LIN {X 0,Y 523.484,Z 545.078,A -85,B 0,C 180,E1 -4763.834,E2 -4763.834} C_VEL
LIN {X 0,Y 523.383,Z 549.826,A -85,B 0,C 180,E1 -4764.992,E2 -4764.992} C_VEL
LIN {X 0,Y 523.443,Z 553.457,A -85,B 0,C 180,E1 -4766.15,E2 -4766.15} C_VEL
LIN {X 0,Y 523.367,Z 555.329,A -85,B 0,C 180,E1 -4766.921,E2 -4766.921} C_VEL
LIN {X 0,Y 523.334,Z 556.731,A -85,B 0,C 180,E1 -4767.691,E2 -4767.691} C_VEL
LIN {X 0,Y 523.25,Z 558.341,A -85,B 0,C 180,E1 -4769.23,E2 -4769.23} C_VEL
LIN {X 0,Y 523.25,Z 558.562,A -85,B 0,C 180,E1 -4770,E2 -4770} C_VEL
LIN {X 0,Y 523.274,Z 557.74,A -85,B 0,C 180,E1 -4771.539,E2 -4771.539} C_VEL
LIN {X 0,Y 523.334,Z 556.745,A -85,B 0,C 180,E1 -4772.308,E2 -4772.308} C_VEL
LIN {X 0,Y 523.367,Z 555.347,A -85,B 0,C 180,E1 -4773.079,E2 -4773.079} C_VEL
LIN {X 0,Y 523.424,Z 552.405,A -85,B 0,C 180,E1 -4774.235,E2 -4774.235} C_VEL
LIN {X 0,Y 523.461,Z 548.419,A -85,B 0,C 180,E1 -4775.392,E2 -4775.392} C_VEL
LIN {X 0,Y 523.514,Z 543.187,A -85,B 0,C 180,E1 -4776.572,E2 -4776.572} C_VEL
LIN {X 0,Y 523.638,Z 536.823,A -85,B 0,C 180,E1 -4777.713,E2 -4777.713} C_VEL
LIN {X 0,Y 523.814,Z 528.761,A -85,B 0,C 180,E1 -4778.875,E2 -4778.875} C_VEL
LIN {X 0,Y 524.041,Z 520.543,A -85,B 0,C 180,E1 -4779.845,E2 -4779.845} C_VEL
LIN {X 0,Y 524.298,Z 510.517,A -85,B 0,C 180,E1 -4780.816,E2 -4780.816} C_VEL
LIN {X 0,Y 524.6,Z 499.164,A -85,B 0,C 180,E1 -4781.691,E2 -4781.691} C_VEL
LIN {X 0,Y 524.837,Z 488.067,A -85,B 0,C 180,E1 -4782.371,E2 -4782.371} C_VEL
LIN {X 0,Y 525.075,Z 475.733,A -85,B 0,C 180,E1 -4782.955,E2 -4782.955} C_VEL
LIN {X 0,Y 525.31,Z 462.663,A -85,B 0,C 180,E1 -4783.392,E2 -4783.392} C_VEL
LIN {X 0,Y 525.513,Z 450.182,A -85,B 0,C 180,E1 -4783.658,E2 -4783.658} C_VEL
LIN {X 0,Y 525.797,Z 355.668,A -85,B 0,C 180,E1 -4784.969,E2 -4784.969} C_VEL
LIN {X 0,Y 524.316,Z 345.731,A -85,B 0,C 180,E1 -4785.168,E2 -4785.168} C_VEL
LIN {X 0,Y 524.755,Z 323.816,A -85,B 0,C 180,E1 -4788.526,E2 -4788.526} C_VEL
LIN {X 0,Y 525.188,Z 305.323,A -85,B 0,C 180,E1 -4791.386,E2 -4791.386} C_VEL
LIN {X 0,Y 525.479,Z 293.613,A -85,B 0,C 180,E1 -4793.237,E2 -4793.237} C_VEL
LIN {X 0,Y 523.982,Z 285.216,A -85,B 0,C 180,E1 -4794.674,E2 -4794.674} C_VEL
LIN {X 0,Y 523.978,Z 285.218,A -85,B 0,C 180,E1 -4797.718,E2 -4797.718} C_VEL
LIN {X 0,Y 523.943,Z 285.215,A -85,B 0,C 180,E1 -4800.854,E2 -4800.854} C_VEL
LIN {X 0,Y 523.957,Z 285.216,A -85,B 0,C 180,E1 -4803.734,E2 -4803.734} C_VEL
LIN {X 0,Y 523.901,Z 285.227,A -85,B 0,C 180,E1 -4806.401,E2 -4806.401} C_VEL
LIN {X 0,Y 523.917,Z 285.218,A -85,B 0,C 180,E1 -4809.084,E2 -4809.084} C_VEL
LIN {X 0,Y 523.952,Z 285.218,A -85,B 0,C 180,E1 -4812.118,E2 -4812.118} C_VEL
LIN {X 0,Y 523.952,Z 285.213,A -85,B 0,C 180,E1 -4815.308,E2 -4815.308} C_VEL
LIN {X 0,Y 523.958,Z 285.221,A -85,B 0,C 180,E1 -4818.688,E2 -4818.688} C_VEL
LIN {X 0,Y 523.915,Z 285.218,A -85,B 0,C 180,E1 -4821.898,E2 -4821.898} C_VEL
LIN {X 0,Y 523.93,Z 285.224,A -85,B 0,C 180,E1 -4824.909,E2 -4824.909} C_VEL
LIN {X 0,Y 523.938,Z 285.215,A -85,B 0,C 180,E1 -4827.678,E2 -4827.678} C_VEL
LIN {X 0,Y 523.949,Z 285.219,A -85,B 0,C 180,E1 -4830.676,E2 -4830.676} C_VEL
LIN {X 0,Y 523.969,Z 285.212,A -85,B 0,C 180,E1 -4833.728,E2 -4833.728} C_VEL
LIN {X 0,Y 523.931,Z 285.216,A -85,B 0,C 180,E1 -4836.271,E2 -4836.271} C_VEL
LIN {X 0,Y 523.94,Z 285.219,A -85,B 0,C 180,E1 -4838.766,E2 -4838.766} C_VEL
LIN {X 0,Y 523.946,Z 285.224,A -85,B 0,C 180,E1 -4841.221,E2 -4841.221} C_VEL
LIN {X 0,Y 523.931,Z 285.22,A -85,B 0,C 180,E1 -4843.639,E2 -4843.639} C_VEL
LIN {X 0,Y 523.939,Z 285.216,A -85,B 0,C 180,E1 -4846.028,E2 -4846.028} C_VEL
LIN {X 0,Y 524.006,Z 285.206,A -85,B 0,C 180,E1 -4848.394,E2 -4848.394} C_VEL
LIN {X 0,Y 523.999,Z 285.217,A -85,B 0,C 180,E1 -4851.516,E2 -4851.516} C_VEL
LIN {X 0,Y 524.077,Z 285.198,A -85,B 0,C 180,E1 -4854.614,E2 -4854.614} C_VEL
LIN {X 0,Y 524.103,Z 285.204,A -85,B 0,C 180,E1 -4857.695,E2 -4857.695} C_VEL
LIN {X 0,Y 524.116,Z 285.193,A -85,B 0,C 180,E1 -4860.769,E2 -4860.769} C_VEL
LIN {X 0,Y 524.067,Z 285.2,A -85,B 0,C 180,E1 -4863.075,E2 -4863.075} C_VEL
LIN {X 0,Y 524.023,Z 285.21,A -85,B 0,C 180,E1 -4866.16,E2 -4866.16} C_VEL
LIN {X 0,Y 523.998,Z 285.21,A -85,B 0,C 180,E1 -4868.484,E2 -4868.484} C_VEL
LIN {X 0,Y 523.997,Z 285.213,A -85,B 0,C 180,E1 -4871.74,E2 -4871.74} C_VEL
LIN {X 0,Y 523.986,Z 285.209,A -85,B 0,C 180,E1 -4875.052,E2 -4875.052} C_VEL
LIN {X 0,Y 523.942,Z 285.22,A -85,B 0,C 180,E1 -4877.97,E2 -4877.97} C_VEL
LIN {X 0,Y 523.967,Z 285.219,A -85,B 0,C 180,E1 -4880.411,E2 -4880.411} C_VEL
LIN {X 0,Y 523.905,Z 285.221,A -85,B 0,C 180,E1 -4882.894,E2 -4882.894} C_VEL
LIN {X 0,Y 523.925,Z 285.216,A -85,B 0,C 180,E1 -4885.42,E2 -4885.42} C_VEL
LIN {X 0,Y 523.913,Z 285.221,A -85,B 0,C 180,E1 -4888.003,E2 -4888.003} C_VEL
LIN {X 0,Y 523.94,Z 285.22,A -85,B 0,C 180,E1 -4890.855,E2 -4890.855} C_VEL
LIN {X 0,Y 523.955,Z 285.213,A -85,B 0,C 180,E1 -4893.735,E2 -4893.735} C_VEL
LIN {X 0,Y 523.9,Z 285.225,A -85,B 0,C 180,E1 -4896.402,E2 -4896.402} C_VEL
LIN {X 0,Y 523.91,Z 285.223,A -85,B 0,C 180,E1 -4899.086,E2 -4899.086} C_VEL
LIN {X 0,Y 523.935,Z 285.216,A -85,B 0,C 180,E1 -4902.121,E2 -4902.121} C_VEL
LIN {X 0,Y 523.938,Z 285.219,A -85,B 0,C 180,E1 -4905.311,E2 -4905.311} C_VEL
LIN {X 0,Y 523.894,Z 285.227,A -85,B 0,C 180,E1 -4906.894,E2 -4906.894} C_VEL
LIN {X 0,Y 523.214,Z 285.308,A -85,B 0,C 180,E1 -4907.535,E2 -4907.535} C_VEL
LIN {X 0,Y 520.363,Z 285.663,A -85,B 0,C 180,E1 -4908.577,E2 -4908.577} C_VEL
LIN {X 0,Y 517.964,Z 285.963,A -85,B 0,C 180,E1 -4909.416,E2 -4909.416} C_VEL
LIN {X 0,Y 516.939,Z 286.087,A -85,B 0,C 180,E1 -4910.063,E2 -4910.063} C_VEL
LIN {X 0,Y 516.857,Z 286.097,A -85,B 0,C 180,E1 -4910.283,E2 -4910.283} C_VEL
LIN {X 0,Y 516.874,Z 286.104,A -85,B 0,C 180,E1 -4913.255,E2 -4913.255} C_VEL
LIN {X 0,Y 516.884,Z 286.094,A -85,B 0,C 180,E1 -4916.12,E2 -4916.12} C_VEL
LIN {X 0,Y 516.88,Z 286.098,A -85,B 0,C 180,E1 -4918.939,E2 -4918.939} C_VEL
LIN {X 0,Y 516.849,Z 286.105,A -85,B 0,C 180,E1 -4921.581,E2 -4921.581} C_VEL
LIN {X 0,Y 516.86,Z 286.097,A -85,B 0,C 180,E1 -4924.208,E2 -4924.208} C_VEL
LIN {X 0,Y 516.859,Z 286.097,A -85,B 0,C 180,E1 -4926.777,E2 -4926.777} C_VEL
LIN {X 0,Y 516.933,Z 286.096,A -85,B 0,C 180,E1 -4929.735,E2 -4929.735} C_VEL
LIN {X 0,Y 516.887,Z 286.093,A -85,B 0,C 180,E1 -4932.595,E2 -4932.595} C_VEL
LIN {X 0,Y 516.946,Z 286.087,A -85,B 0,C 180,E1 -4935.031,E2 -4935.031} C_VEL
LIN {X 0,Y 516.93,Z 286.092,A -85,B 0,C 180,E1 -4938.233,E2 -4938.233} C_VEL
LIN {X 0,Y 516.923,Z 286.091,A -85,B 0,C 180,E1 -4941.399,E2 -4941.399} C_VEL
LIN {X 0,Y 516.983,Z 286.084,A -85,B 0,C 180,E1 -4944.54,E2 -4944.54} C_VEL
LIN {X 0,Y 517.071,Z 286.073,A -85,B 0,C 180,E1 -4947.664,E2 -4947.664} C_VEL
LIN {X 0,Y 517.068,Z 286.078,A -85,B 0,C 180,E1 -4950,E2 -4950} C_VEL
LIN {X 0,Y 517.069,Z 286.079,A -85,B 0,C 180,E1 -4952.337,E2 -4952.337} C_VEL
LIN {X 0,Y 516.972,Z 286.091,A -85,B 0,C 180,E1 -4956.244,E2 -4956.244} C_VEL
LIN {X 0,Y 516.902,Z 286.091,A -85,B 0,C 180,E1 -4959.391,E2 -4959.391} C_VEL
LIN {X 0,Y 516.882,Z 286.103,A -85,B 0,C 180,E1 -4962.566,E2 -4962.566} C_VEL
LIN {X 0,Y 516.837,Z 286.1,A -85,B 0,C 180,E1 -4965.781,E2 -4965.781} C_VEL
LIN {X 0,Y 516.874,Z 286.098,A -85,B 0,C 180,E1 -4968.224,E2 -4968.224} C_VEL
LIN {X 0,Y 516.882,Z 286.103,A -85,B 0,C 180,E1 -4970.703,E2 -4970.703} C_VEL
LIN {X 0,Y 516.848,Z 286.104,A -85,B 0,C 180,E1 -4973.225,E2 -4973.225} C_VEL
LIN {X 0,Y 516.856,Z 286.102,A -85,B 0,C 180,E1 -4976.175,E2 -4976.175} C_VEL
LIN {X 0,Y 516.912,Z 286.308,A -85,B 0,C 180,E1 -4977.15,E2 -4977.15} C_VEL
LIN {X 0,Y 517.552,Z 290.673,A -85,B 0,C 180,E1 -4978.035,E2 -4978.035} C_VEL
LIN {X 0,Y 517.288,Z 305.162,A -85,B 0,C 180,E1 -4980.856,E2 -4980.856} C_VEL
LIN {X 0,Y 517.209,Z 309.487,A -85,B 0,C 180,E1 -4981.687,E2 -4981.687} C_VEL
LIN {X 0,Y 519.12,Z 321.055,A -85,B 0,C 180,E1 -4981.925,E2 -4981.925} C_VEL
LIN {X 0,Y 518.626,Z 416.658,A -85,B 0,C 180,E1 -4983.288,E2 -4983.288} C_VEL
LIN {X 0,Y 518.388,Z 430.021,A -85,B 0,C 180,E1 -4983.641,E2 -4983.641} C_VEL
LIN {X 0,Y 518.174,Z 441.438,A -85,B 0,C 180,E1 -4984.086,E2 -4984.086} C_VEL
LIN {X 0,Y 517.884,Z 452.681,A -85,B 0,C 180,E1 -4984.668,E2 -4984.668} C_VEL
LIN {X 0,Y 517.613,Z 463.334,A -85,B 0,C 180,E1 -4985.369,E2 -4985.369} C_VEL
LIN {X 0,Y 517.364,Z 473.747,A -85,B 0,C 180,E1 -4986.222,E2 -4986.222} C_VEL
LIN {X 0,Y 517.004,Z 484.69,A -85,B 0,C 180,E1 -4987.346,E2 -4987.346} C_VEL
LIN {X 0,Y 516.8,Z 492.236,A -85,B 0,C 180,E1 -4988.305,E2 -4988.305} C_VEL
LIN {X 0,Y 516.619,Z 499.468,A -85,B 0,C 180,E1 -4989.426,E2 -4989.426} C_VEL
LIN {X 0,Y 516.474,Z 504.474,A -85,B 0,C 180,E1 -4990.356,E2 -4990.356} C_VEL
LIN {X 0,Y 516.39,Z 509.598,A -85,B 0,C 180,E1 -4991.535,E2 -4991.535} C_VEL
LIN {X 0,Y 516.329,Z 513.522,A -85,B 0,C 180,E1 -4992.69,E2 -4992.69} C_VEL
LIN {X 0,Y 516.259,Z 516.694,A -85,B 0,C 180,E1 -4993.97,E2 -4993.97} C_VEL
LIN {X 0,Y 516.213,Z 518.527,A -85,B 0,C 180,E1 -4995.069,E2 -4995.069} C_VEL
LIN {X 0,Y 516.184,Z 519.573,A -85,B 0,C 180,E1 -4996.188,E2 -4996.188} C_VEL
LIN {X 0,Y 516.178,Z 519.794,A -85,B 0,C 180,E1 -4997.327,E2 -4997.327} C_VEL
LIN {X 0,Y 516.197,Z 519.147,A -85,B 0,C 180,E1 -4998.489,E2 -4998.489} C_VEL
LIN {X 0,Y 516.196,Z 517.568,A -85,B 0,C 180,E1 -4999.68,E2 -4999.68} C_VEL
LIN {X 0,Y 516.287,Z 514.031,A -85,B 0,C 180,E1 -5001.231,E2 -5001.231} C_VEL
LIN {X 0,Y 516.386,Z 510.828,A -85,B 0,C 180,E1 -5002.233,E2 -5002.233} C_VEL
LIN {X 0,Y 516.471,Z 506.049,A -85,B 0,C 180,E1 -5003.404,E2 -5003.404} C_VEL
LIN {X 0,Y 516.586,Z 500.555,A -85,B 0,C 180,E1 -5004.483,E2 -5004.483} C_VEL
LIN {X 0,Y 516.783,Z 493.342,A -85,B 0,C 180,E1 -5005.634,E2 -5005.634} C_VEL
LIN {X 0,Y 517.017,Z 485.983,A -85,B 0,C 180,E1 -5006.596,E2 -5006.596} C_VEL
LIN {X 0,Y 517.277,Z 476.668,A -85,B 0,C 180,E1 -5007.603,E2 -5007.603} C_VEL
LIN {X 0,Y 517.538,Z 465.559,A -85,B 0,C 180,E1 -5008.562,E2 -5008.562} C_VEL
LIN {X 0,Y 517.86,Z 454.909,A -85,B 0,C 180,E1 -5009.295,E2 -5009.295} C_VEL
LIN {X 0,Y 518.163,Z 442.997,A -85,B 0,C 180,E1 -5009.935,E2 -5009.935} C_VEL
LIN {X 0,Y 518.359,Z 430.294,A -85,B 0,C 180,E1 -5010.442,E2 -5010.442} C_VEL
LIN {X 0,Y 518.56,Z 416.327,A -85,B 0,C 180,E1 -5010.811,E2 -5010.811} C_VEL
LIN {X 0,Y 518.973,Z 319.058,A -85,B 0,C 180,E1 -5012.201,E2 -5012.201} C_VEL
LIN {X 0,Y 517.197,Z 309.037,A -85,B 0,C 180,E1 -5012.401,E2 -5012.401} C_VEL
LIN {X 0,Y 517.21,Z 289.506,A -85,B 0,C 180,E1 -5015.666,E2 -5015.666} C_VEL
LIN {X 0,Y 516.991,Z 286.087,A -85,B 0,C 180,E1 -5016.251,E2 -5016.251} C_VEL
LIN {X 0,Y 516.942,Z 286.092,A -85,B 0,C 180,E1 -5019.731,E2 -5019.731} C_VEL
LIN {X 0,Y 516.909,Z 286.095,A -85,B 0,C 180,E1 -5022.595,E2 -5022.595} C_VEL
LIN {X 0,Y 516.954,Z 286.092,A -85,B 0,C 180,E1 -5025.03,E2 -5025.03} C_VEL
LIN {X 0,Y 516.968,Z 286.085,A -85,B 0,C 180,E1 -5028.233,E2 -5028.233} C_VEL
LIN {X 0,Y 516.964,Z 286.091,A -85,B 0,C 180,E1 -5031.399,E2 -5031.399} C_VEL
LIN {X 0,Y 517.003,Z 286.088,A -85,B 0,C 180,E1 -5033.757,E2 -5033.757} C_VEL
LIN {X 0,Y 517.013,Z 286.079,A -85,B 0,C 180,E1 -5036.883,E2 -5036.883} C_VEL
LIN {X 0,Y 517.087,Z 286.077,A -85,B 0,C 180,E1 -5040,E2 -5040} C_VEL
LIN {X 0,Y 517.013,Z 286.078,A -85,B 0,C 180,E1 -5043.117,E2 -5043.117} C_VEL
LIN {X 0,Y 516.989,Z 286.087,A -85,B 0,C 180,E1 -5046.243,E2 -5046.243} C_VEL
LIN {X 0,Y 516.967,Z 286.087,A -85,B 0,C 180,E1 -5048.6,E2 -5048.6} C_VEL
LIN {X 0,Y 516.953,Z 286.088,A -85,B 0,C 180,E1 -5051.807,E2 -5051.807} C_VEL
LIN {X 0,Y 516.949,Z 286.087,A -85,B 0,C 180,E1 -5055.147,E2 -5055.147} C_VEL
LIN {X 0,Y 516.917,Z 286.093,A -85,B 0,C 180,E1 -5058.222,E2 -5058.222} C_VEL
LIN {X 0,Y 516.914,Z 286.096,A -85,B 0,C 180,E1 -5060.701,E2 -5060.701} C_VEL
LIN {X 0,Y 516.904,Z 286.092,A -85,B 0,C 180,E1 -5064.072,E2 -5064.072} C_VEL
LIN {X 0,Y 516.925,Z 286.096,A -85,B 0,C 180,E1 -5066.658,E2 -5066.658} C_VEL
LIN {X 0,Y 516.912,Z 286.092,A -85,B 0,C 180,E1 -5069.524,E2 -5069.524} C_VEL
LIN {X 0,Y 516.895,Z 286.095,A -85,B 0,C 180,E1 -5072.543,E2 -5072.543} C_VEL
LIN {X 0,Y 516.867,Z 286.103,A -85,B 0,C 180,E1 -5075.329,E2 -5075.329} C_VEL
LIN {X 0,Y 516.882,Z 286.094,A -85,B 0,C 180,E1 -5077.943,E2 -5077.943} C_VEL
LIN {X 0,Y 516.885,Z 286.096,A -85,B 0,C 180,E1 -5080.742,E2 -5080.742} C_VEL
LIN {X 0,Y 516.884,Z 286.098,A -85,B 0,C 180,E1 -5082.831,E2 -5082.831} C_VEL
LIN {X 0,Y 516.897,Z 286.097,A -85,B 0,C 180,E1 -5085.007,E2 -5085.007} C_VEL
LIN {X 0,Y 516.915,Z 286.091,A -85,B 0,C 180,E1 -5088.399,E2 -5088.399} C_VEL
LIN {X 0,Y 516.882,Z 286.1,A -85,B 0,C 180,E1 -5091.284,E2 -5091.284} C_VEL
LIN {X 0,Y 516.873,Z 286.101,A -85,B 0,C 180,E1 -5094.22,E2 -5094.22} C_VEL
LIN {X 0,Y 516.897,Z 286.097,A -85,B 0,C 180,E1 -5097.053,E2 -5097.053} C_VEL
LIN {X 0,Y 516.895,Z 286.102,A -85,B 0,C 180,E1 -5099.796,E2 -5099.796} C_VEL
LIN {X 0,Y 516.927,Z 286.095,A -85,B 0,C 180,E1 -5102.467,E2 -5102.467} C_VEL
LIN {X 0,Y 516.908,Z 286.098,A -85,B 0,C 180,E1 -5105.396,E2 -5105.396} C_VEL
LIN {X 0,Y 516.921,Z 286.184,A -85,B 0,C 180,E1 -5105.518,E2 -5105.518} C_VEL
LIN {X 0,Y 518.271,Z 294.325,A -85,B 0,C 180,E1 -5106.843,E2 -5106.843} C_VEL
LIN {X 0,Y 517.895,Z 313.462,A -85,B 0,C 180,E1 -5109.794,E2 -5109.794} C_VEL
LIN {X 0,Y 517.504,Z 331.908,A -85,B 0,C 180,E1 -5112.616,E2 -5112.616} C_VEL
LIN {X 0,Y 517.251,Z 345.235,A -85,B 0,C 180,E1 -5114.634,E2 -5114.634} C_VEL
LIN {X 0,Y 519.038,Z 358.299,A -85,B 0,C 180,E1 -5114.876,E2 -5114.876} C_VEL
LIN {X 0,Y 518.533,Z 453.585,A -85,B 0,C 180,E1 -5116.229,E2 -5116.229} C_VEL
LIN {X 0,Y 518.3,Z 466.903,A -85,B 0,C 180,E1 -5116.572,E2 -5116.572} C_VEL
LIN {X 0,Y 518.025,Z 479.679,A -85,B 0,C 180,E1 -5117.064,E2 -5117.064} C_VEL
LIN {X 0,Y 517.775,Z 491.966,A -85,B 0,C 180,E1 -5117.713,E2 -5117.713} C_VEL
LIN {X 0,Y 517.486,Z 504.066,A -85,B 0,C 180,E1 -5118.543,E2 -5118.543} C_VEL
LIN {X 0,Y 517.159,Z 514.372,A -85,B 0,C 180,E1 -5119.428,E2 -5119.428} C_VEL
LIN {X 0,Y 516.89,Z 523.628,A -85,B 0,C 180,E1 -5120.412,E2 -5120.412} C_VEL
LIN {X 0,Y 516.656,Z 532.638,A -85,B 0,C 180,E1 -5121.591,E2 -5121.591} C_VEL
LIN {X 0,Y 516.505,Z 539.895,A -85,B 0,C 180,E1 -5122.769,E2 -5122.769} C_VEL
LIN {X 0,Y 516.397,Z 544.787,A -85,B 0,C 180,E1 -5123.749,E2 -5123.749} C_VEL
LIN {X 0,Y 516.313,Z 549.544,A -85,B 0,C 180,E1 -5124.924,E2 -5124.924} C_VEL
LIN {X 0,Y 516.352,Z 553.181,A -85,B 0,C 180,E1 -5126.097,E2 -5126.097} C_VEL
LIN {X 0,Y 516.282,Z 555.056,A -85,B 0,C 180,E1 -5126.878,E2 -5126.878} C_VEL
LIN {X 0,Y 516.26,Z 556.462,A -85,B 0,C 180,E1 -5127.659,E2 -5127.659} C_VEL
LIN {X 0,Y 516.16,Z 558.076,A -85,B 0,C 180,E1 -5129.219,E2 -5129.219} C_VEL
LIN {X 0,Y 516.158,Z 558.298,A -85,B 0,C 180,E1 -5130,E2 -5130} C_VEL
LIN {X 0,Y 516.191,Z 557.476,A -85,B 0,C 180,E1 -5131.56,E2 -5131.56} C_VEL
LIN {X 0,Y 516.26,Z 556.482,A -85,B 0,C 180,E1 -5132.34,E2 -5132.34} C_VEL
LIN {X 0,Y 516.282,Z 555.082,A -85,B 0,C 180,E1 -5133.121,E2 -5133.121} C_VEL
LIN {X 0,Y 516.311,Z 552.137,A -85,B 0,C 180,E1 -5134.293,E2 -5134.293} C_VEL
LIN {X 0,Y 516.375,Z 548.148,A -85,B 0,C 180,E1 -5135.466,E2 -5135.466} C_VEL
LIN {X 0,Y 516.45,Z 542.212,A -85,B 0,C 180,E1 -5136.798,E2 -5136.798} C_VEL
LIN {X 0,Y 516.594,Z 535.298,A -85,B 0,C 180,E1 -5138.015,E2 -5138.015} C_VEL
LIN {X 0,Y 516.791,Z 526.97,A -85,B 0,C 180,E1 -5139.194,E2 -5139.194} C_VEL
LIN {X 0,Y 517.024,Z 518.423,A -85,B 0,C 180,E1 -5140.178,E2 -5140.178} C_VEL
LIN {X 0,Y 517.365,Z 507.866,A -85,B 0,C 180,E1 -5141.161,E2 -5141.161} C_VEL
LIN {X 0,Y 517.668,Z 496.325,A -85,B 0,C 180,E1 -5142.024,E2 -5142.024} C_VEL
LIN {X 0,Y 517.915,Z 485.935,A -85,B 0,C 180,E1 -5142.639,E2 -5142.639} C_VEL
LIN {X 0,Y 518.169,Z 474.071,A -85,B 0,C 180,E1 -5143.181,E2 -5143.181} C_VEL
LIN {X 0,Y 518.46,Z 460.393,A -85,B 0,C 180,E1 -5143.622,E2 -5143.622} C_VEL
LIN {X 0,Y 518.624,Z 448.136,A -85,B 0,C 180,E1 -5143.868,E2 -5143.868} C_VEL
LIN {X 0,Y 518.974,Z 356.531,A -85,B 0,C 180,E1 -5145.154,E2 -5145.154} C_VEL
LIN {X 0,Y 517.291,Z 345.567,A -85,B 0,C 180,E1 -5145.366,E2 -5145.366} C_VEL
LIN {X 0,Y 517.815,Z 323.455,A -85,B 0,C 180,E1 -5148.804,E2 -5148.804} C_VEL
LIN {X 0,Y 518.26,Z 305.148,A -85,B 0,C 180,E1 -5151.686,E2 -5151.686} C_VEL
LIN {X 0,Y 518.511,Z 294.727,A -85,B 0,C 180,E1 -5153.356,E2 -5153.356} C_VEL
LIN {X 0,Y 516.941,Z 286.093,A -85,B 0,C 180,E1 -5154.855,E2 -5154.855} C_VEL
LIN {X 0,Y 516.926,Z 286.097,A -85,B 0,C 180,E1 -5157.905,E2 -5157.905} C_VEL
LIN {X 0,Y 516.891,Z 286.101,A -85,B 0,C 180,E1 -5160.203,E2 -5160.203} C_VEL
LIN {X 0,Y 516.893,Z 286.093,A -85,B 0,C 180,E1 -5162.946,E2 -5162.946} C_VEL
LIN {X 0,Y 516.869,Z 286.098,A -85,B 0,C 180,E1 -5165.78,E2 -5165.78} C_VEL
LIN {X 0,Y 516.878,Z 286.098,A -85,B 0,C 180,E1 -5168.715,E2 -5168.715} C_VEL
LIN {X 0,Y 516.911,Z 286.092,A -85,B 0,C 180,E1 -5171.774,E2 -5171.774} C_VEL
LIN {X 0,Y 516.919,Z 286.092,A -85,B 0,C 180,E1 -5175.01,E2 -5175.01} C_VEL
LIN {X 0,Y 516.914,Z 286.097,A -85,B 0,C 180,E1 -5178.398,E2 -5178.398} C_VEL
LIN {X 0,Y 516.879,Z 286.096,A -85,B 0,C 180,E1 -5181.284,E2 -5181.284} C_VEL
LIN {X 0,Y 516.883,Z 286.096,A -85,B 0,C 180,E1 -5184.221,E2 -5184.221} C_VEL
LIN {X 0,Y 516.893,Z 286.099,A -85,B 0,C 180,E1 -5187.053,E2 -5187.053} C_VEL
LIN {X 0,Y 516.888,Z 286.093,A -85,B 0,C 180,E1 -5189.796,E2 -5189.796} C_VEL
LIN {X 0,Y 516.923,Z 286.091,A -85,B 0,C 180,E1 -5192.467,E2 -5192.467} C_VEL
LIN {X 0,Y 516.905,Z 286.101,A -85,B 0,C 180,E1 -5195.072,E2 -5195.072} C_VEL
LIN {X 0,Y 516.864,Z 286.099,A -85,B 0,C 180,E1 -5197.621,E2 -5197.621} C_VEL
LIN {X 0,Y 516.926,Z 286.088,A -85,B 0,C 180,E1 -5200.13,E2 -5200.13} C_VEL
LIN {X 0,Y 516.923,Z 286.09,A -85,B 0,C 180,E1 -5202.596,E2 -5202.596} C_VEL
LIN {X 0,Y 516.945,Z 286.091,A -85,B 0,C 180,E1 -5205.03,E2 -5205.03} C_VEL
LIN {X 0,Y 516.959,Z 286.085,A -85,B 0,C 180,E1 -5208.234,E2 -5208.234} C_VEL
LIN {X 0,Y 516.964,Z 286.092,A -85,B 0,C 180,E1 -5211.4,E2 -5211.4} C_VEL
LIN {X 0,Y 517.003,Z 286.085,A -85,B 0,C 180,E1 -5213.757,E2 -5213.757} C_VEL
LIN {X 0,Y 517.076,Z 286.08,A -85,B 0,C 180,E1 -5217.663,E2 -5217.663} C_VEL
LIN {X 0,Y 517.086,Z 286.068,A -85,B 0,C 180,E1 -5220.779,E2 -5220.779} C_VEL
LIN {X 0,Y 517.008,Z 286.079,A -85,B 0,C 180,E1 -5223.117,E2 -5223.117} C_VEL
LIN {X 0,Y 516.985,Z 286.085,A -85,B 0,C 180,E1 -5226.244,E2 -5226.244} C_VEL
LIN {X 0,Y 516.963,Z 286.085,A -85,B 0,C 180,E1 -5228.601,E2 -5228.601} C_VEL
LIN {X 0,Y 516.946,Z 286.092,A -85,B 0,C 180,E1 -5231.807,E2 -5231.807} C_VEL
LIN {X 0,Y 516.938,Z 286.087,A -85,B 0,C 180,E1 -5235.146,E2 -5235.146} C_VEL
LIN {X 0,Y 516.91,Z 286.101,A -85,B 0,C 180,E1 -5238.223,E2 -5238.223} C_VEL
LIN {X 0,Y 516.907,Z 286.094,A -85,B 0,C 180,E1 -5240.702,E2 -5240.702} C_VEL
LIN {X 0,Y 516.885,Z 286.098,A -85,B 0,C 180,E1 -5244.074,E2 -5244.074} C_VEL
LIN {X 0,Y 516.893,Z 286.099,A -85,B 0,C 180,E1 -5246.66,E2 -5246.66} C_VEL
LIN {X 0,Y 516.906,Z 286.091,A -85,B 0,C 180,E1 -5249.524,E2 -5249.524} C_VEL
LIN {X 0,Y 516.892,Z 286.102,A -85,B 0,C 180,E1 -5252.544,E2 -5252.544} C_VEL
LIN {X 0,Y 516.862,Z 286.098,A -85,B 0,C 180,E1 -5255.33,E2 -5255.33} C_VEL
LIN {X 0,Y 516.876,Z 286.095,A -85,B 0,C 180,E1 -5257.944,E2 -5257.944} C_VEL
LIN {X 0,Y 516.87,Z 286.104,A -85,B 0,C 180,E1 -5260.744,E2 -5260.744} C_VEL
LIN {X 0,Y 516.852,Z 286.107,A -85,B 0,C 180,E1 -5262.835,E2 -5262.835} C_VEL
LIN {X 0,Y 516.893,Z 286.102,A -85,B 0,C 180,E1 -5265.008,E2 -5265.008} C_VEL
LIN {X 0,Y 516.887,Z 286.095,A -85,B 0,C 180,E1 -5268.403,E2 -5268.403} C_VEL
LIN {X 0,Y 516.857,Z 286.097,A -85,B 0,C 180,E1 -5270.283,E2 -5270.283} C_VEL
LIN {X 0,Y 516.196,Z 286.187,A -85,B 0,C 180,E1 -5270.933,E2 -5270.933} C_VEL
LIN {X 0,Y 513.349,Z 286.542,A -85,B 0,C 180,E1 -5271.989,E2 -5271.989} C_VEL
LIN {X 0,Y 510.935,Z 286.842,A -85,B 0,C 180,E1 -5272.839,E2 -5272.839} C_VEL
LIN {X 0,Y 509.894,Z 286.97,A -85,B 0,C 180,E1 -5273.496,E2 -5273.496} C_VEL
LIN {X 0,Y 509.806,Z 286.978,A -85,B 0,C 180,E1 -5273.718,E2 -5273.718} C_VEL
LIN {X 0,Y 509.841,Z 286.972,A -85,B 0,C 180,E1 -5276.539,E2 -5276.539} C_VEL
LIN {X 0,Y 509.828,Z 286.983,A -85,B 0,C 180,E1 -5279.334,E2 -5279.334} C_VEL
LIN {X 0,Y 509.833,Z 286.973,A -85,B 0,C 180,E1 -5282.052,E2 -5282.052} C_VEL
LIN {X 0,Y 509.797,Z 286.977,A -85,B 0,C 180,E1 -5284.7,E2 -5284.7} C_VEL
LIN {X 0,Y 509.828,Z 286.981,A -85,B 0,C 180,E1 -5287.459,E2 -5287.459} C_VEL
LIN {X 0,Y 509.909,Z 286.969,A -85,B 0,C 180,E1 -5289.845,E2 -5289.845} C_VEL
LIN {X 0,Y 509.855,Z 286.971,A -85,B 0,C 180,E1 -5293.174,E2 -5293.174} C_VEL
LIN {X 0,Y 509.862,Z 286.976,A -85,B 0,C 180,E1 -5295.635,E2 -5295.635} C_VEL
LIN {X 0,Y 509.893,Z 286.97,A -85,B 0,C 180,E1 -5298.131,E2 -5298.131} C_VEL
LIN {X 0,Y 509.876,Z 286.968,A -85,B 0,C 180,E1 -5301.28,E2 -5301.28} C_VEL
LIN {X 0,Y 509.922,Z 286.965,A -85,B 0,C 180,E1 -5303.67,E2 -5303.67} C_VEL
LIN {X 0,Y 509.865,Z 286.969,A -85,B 0,C 180,E1 -5306.84,E2 -5306.84} C_VEL
LIN {X 0,Y 509.925,Z 286.966,A -85,B 0,C 180,E1 -5308.421,E2 -5308.421} C_VEL
LIN {X 0,Y 510.037,Z 286.954,A -85,B 0,C 180,E1 -5310,E2 -5310} C_VEL
LIN {X 0,Y 510.037,Z 286.954,A -85,B 0,C 180,E1 -5312.37,E2 -5312.37} C_VEL
LIN {X 0,Y 509.937,Z 286.959,A -85,B 0,C 180,E1 -5315.537,E2 -5315.537} C_VEL
LIN {X 0,Y 509.878,Z 286.969,A -85,B 0,C 180,E1 -5317.923,E2 -5317.923} C_VEL
LIN {X 0,Y 509.855,Z 286.97,A -85,B 0,C 180,E1 -5321.127,E2 -5321.127} C_VEL
LIN {X 0,Y 509.818,Z 286.974,A -85,B 0,C 180,E1 -5323.554,E2 -5323.554} C_VEL
LIN {X 0,Y 509.806,Z 286.977,A -85,B 0,C 180,E1 -5326.005,E2 -5326.005} C_VEL
LIN {X 0,Y 509.831,Z 286.979,A -85,B 0,C 180,E1 -5328.485,E2 -5328.485} C_VEL
LIN {X 0,Y 509.828,Z 286.98,A -85,B 0,C 180,E1 -5331.003,E2 -5331.003} C_VEL
LIN {X 0,Y 509.808,Z 286.979,A -85,B 0,C 180,E1 -5333.565,E2 -5333.565} C_VEL
LIN {X 0,Y 509.877,Z 287.108,A -85,B 0,C 180,E1 -5337.002,E2 -5337.002} C_VEL
LIN {X 0,Y 510.589,Z 293.212,A -85,B 0,C 180,E1 -5338.244,E2 -5338.244} C_VEL
LIN {X 0,Y 510.252,Z 309.902,A -85,B 0,C 180,E1 -5341.487,E2 -5341.487} C_VEL
LIN {X 0,Y 512.275,Z 321.605,A -85,B 0,C 180,E1 -5341.723,E2 -5341.723} C_VEL
LIN {X 0,Y 511.738,Z 416.812,A -85,B 0,C 180,E1 -5343.103,E2 -5343.103} C_VEL
LIN {X 0,Y 511.494,Z 430.115,A -85,B 0,C 180,E1 -5343.458,E2 -5343.458} C_VEL
LIN {X 0,Y 511.22,Z 442.541,A -85,B 0,C 180,E1 -5343.952,E2 -5343.952} C_VEL
LIN {X 0,Y 510.925,Z 453.715,A -85,B 0,C 180,E1 -5344.548,E2 -5344.548} C_VEL
LIN {X 0,Y 510.652,Z 464.914,A -85,B 0,C 180,E1 -5345.313,E2 -5345.313} C_VEL
LIN {X 0,Y 510.371,Z 474.626,A -85,B 0,C 180,E1 -5346.137,E2 -5346.137} C_VEL
LIN {X 0,Y 510.037,Z 483.99,A -85,B 0,C 180,E1 -5347.106,E2 -5347.106} C_VEL
LIN {X 0,Y 509.761,Z 492.574,A -85,B 0,C 180,E1 -5348.2,E2 -5348.2} C_VEL
LIN {X 0,Y 509.547,Z 500.331,A -85,B 0,C 180,E1 -5349.431,E2 -5349.431} C_VEL
LIN {X 0,Y 509.384,Z 506.426,A -85,B 0,C 180,E1 -5350.637,E2 -5350.637} C_VEL
LIN {X 0,Y 509.3,Z 511.185,A -85,B 0,C 180,E1 -5351.826,E2 -5351.826} C_VEL
LIN {X 0,Y 509.236,Z 514.778,A -85,B 0,C 180,E1 -5352.991,E2 -5352.991} C_VEL
LIN {X 0,Y 509.163,Z 517.357,A -85,B 0,C 180,E1 -5354.13,E2 -5354.13} C_VEL
LIN {X 0,Y 509.119,Z 519.04,A -85,B 0,C 180,E1 -5355.249,E2 -5355.249} C_VEL
LIN {X 0,Y 509.091,Z 519.916,A -85,B 0,C 180,E1 -5356.349,E2 -5356.349} C_VEL
LIN {X 0,Y 509.081,Z 520.039,A -85,B 0,C 180,E1 -5357.432,E2 -5357.432} C_VEL
LIN {X 0,Y 509.105,Z 519.423,A -85,B 0,C 180,E1 -5358.499,E2 -5358.499} C_VEL
LIN {X 0,Y 509.12,Z 518.133,A -85,B 0,C 180,E1 -5359.548,E2 -5359.548} C_VEL
LIN {X 0,Y 509.203,Z 514.781,A -85,B 0,C 180,E1 -5361.115,E2 -5361.115} C_VEL
LIN {X 0,Y 509.311,Z 511.314,A -85,B 0,C 180,E1 -5362.244,E2 -5362.244} C_VEL
LIN {X 0,Y 509.411,Z 506.804,A -85,B 0,C 180,E1 -5363.384,E2 -5363.384} C_VEL
LIN {X 0,Y 509.547,Z 500.745,A -85,B 0,C 180,E1 -5364.599,E2 -5364.599} C_VEL
LIN {X 0,Y 509.771,Z 493.191,A -85,B 0,C 180,E1 -5365.812,E2 -5365.812} C_VEL
LIN {X 0,Y 510.033,Z 484.836,A -85,B 0,C 180,E1 -5366.898,E2 -5366.898} C_VEL
LIN {X 0,Y 510.329,Z 474.45,A -85,B 0,C 180,E1 -5367.98,E2 -5367.98} C_VEL
LIN {X 0,Y 510.631,Z 464.152,A -85,B 0,C 180,E1 -5368.845,E2 -5368.845} C_VEL
LIN {X 0,Y 510.978,Z 452.971,A -85,B 0,C 180,E1 -5369.593,E2 -5369.593} C_VEL
LIN {X 0,Y 511.296,Z 440.828,A -85,B 0,C 180,E1 -5370.219,E2 -5370.219} C_VEL
LIN {X 0,Y 511.49,Z 427.527,A -85,B 0,C 180,E1 -5370.72,E2 -5370.72} C_VEL
LIN {X 0,Y 511.697,Z 414.611,A -85,B 0,C 180,E1 -5371.029,E2 -5371.029} C_VEL
LIN {X 0,Y 512.245,Z 320.538,A -85,B 0,C 180,E1 -5372.388,E2 -5372.388} C_VEL
LIN {X 0,Y 510.2,Z 309.109,A -85,B 0,C 180,E1 -5372.629,E2 -5372.629} C_VEL
LIN {X 0,Y 510.198,Z 291.485,A -85,B 0,C 180,E1 -5375.59,E2 -5375.59} C_VEL
LIN {X 0,Y 509.933,Z 286.967,A -85,B 0,C 180,E1 -5376.36,E2 -5376.36} C_VEL
LIN {X 0,Y 509.919,Z 286.966,A -85,B 0,C 180,E1 -5379.844,E2 -5379.844} C_VEL
LIN {X 0,Y 509.877,Z 286.977,A -85,B 0,C 180,E1 -5383.174,E2 -5383.174} C_VEL
LIN {X 0,Y 509.875,Z 286.977,A -85,B 0,C 180,E1 -5385.634,E2 -5385.634} C_VEL
LIN {X 0,Y 509.915,Z 286.964,A -85,B 0,C 180,E1 -5388.874,E2 -5388.874} C_VEL
LIN {X 0,Y 509.952,Z 286.963,A -85,B 0,C 180,E1 -5392.078,E2 -5392.078} C_VEL
LIN {X 0,Y 509.979,Z 286.956,A -85,B 0,C 180,E1 -5394.464,E2 -5394.464} C_VEL
LIN {X 0,Y 510.055,Z 286.952,A -85,B 0,C 180,E1 -5397.631,E2 -5397.631} C_VEL
LIN {X 0,Y 510.064,Z 286.943,A -85,B 0,C 180,E1 -5400.789,E2 -5400.789} C_VEL
LIN {X 0,Y 509.955,Z 286.958,A -85,B 0,C 180,E1 -5403.16,E2 -5403.16} C_VEL
LIN {X 0,Y 509.937,Z 286.964,A -85,B 0,C 180,E1 -5406.33,E2 -5406.33} C_VEL
LIN {X 0,Y 509.913,Z 286.965,A -85,B 0,C 180,E1 -5408.72,E2 -5408.72} C_VEL
LIN {X 0,Y 509.906,Z 286.967,A -85,B 0,C 180,E1 -5411.931,E2 -5411.931} C_VEL
LIN {X 0,Y 509.896,Z 286.965,A -85,B 0,C 180,E1 -5415.242,E2 -5415.242} C_VEL
LIN {X 0,Y 509.868,Z 286.968,A -85,B 0,C 180,E1 -5417.993,E2 -5417.993} C_VEL
LIN {X 0,Y 509.888,Z 286.973,A -85,B 0,C 180,E1 -5420.401,E2 -5420.401} C_VEL
LIN {X 0,Y 509.831,Z 286.972,A -85,B 0,C 180,E1 -5423.563,E2 -5423.563} C_VEL
LIN {X 0,Y 509.912,Z 286.966,A -85,B 0,C 180,E1 -5426.378,E2 -5426.378} C_VEL
LIN {X 0,Y 509.878,Z 286.973,A -85,B 0,C 180,E1 -5428.844,E2 -5428.844} C_VEL
LIN {X 0,Y 509.821,Z 286.974,A -85,B 0,C 180,E1 -5431.59,E2 -5431.59} C_VEL
LIN {X 0,Y 509.839,Z 286.973,A -85,B 0,C 180,E1 -5434.414,E2 -5434.414} C_VEL
LIN {X 0,Y 509.818,Z 286.98,A -85,B 0,C 180,E1 -5437.341,E2 -5437.341} C_VEL
LIN {X 0,Y 509.84,Z 286.972,A -85,B 0,C 180,E1 -5440.382,E2 -5440.382} C_VEL
LIN {X 0,Y 509.825,Z 286.98,A -85,B 0,C 180,E1 -5443.062,E2 -5443.062} C_VEL
LIN {X 0,Y 509.824,Z 286.978,A -85,B 0,C 180,E1 -5445.793,E2 -5445.793} C_VEL
LIN {X 0,Y 509.857,Z 286.97,A -85,B 0,C 180,E1 -5448.574,E2 -5448.574} C_VEL
LIN {X 0,Y 509.853,Z 286.979,A -85,B 0,C 180,E1 -5451.786,E2 -5451.786} C_VEL
LIN {X 0,Y 509.832,Z 286.976,A -85,B 0,C 180,E1 -5454.622,E2 -5454.622} C_VEL
LIN {X 0,Y 509.864,Z 286.978,A -85,B 0,C 180,E1 -5457.481,E2 -5457.481} C_VEL
LIN {X 0,Y 509.861,Z 286.975,A -85,B 0,C 180,E1 -5460.274,E2 -5460.274} C_VEL
LIN {X 0,Y 509.885,Z 286.971,A -85,B 0,C 180,E1 -5462.944,E2 -5462.944} C_VEL
LIN {X 0,Y 509.898,Z 287.083,A -85,B 0,C 180,E1 -5465.369,E2 -5465.369} C_VEL
LIN {X 0,Y 511.328,Z 296.047,A -85,B 0,C 180,E1 -5466.845,E2 -5466.845} C_VEL
LIN {X 0,Y 510.875,Z 315.534,A -85,B 0,C 180,E1 -5469.884,E2 -5469.884} C_VEL
LIN {X 0,Y 510.44,Z 334.273,A -85,B 0,C 180,E1 -5472.781,E2 -5472.781} C_VEL
LIN {X 0,Y 510.261,Z 344.998,A -85,B 0,C 180,E1 -5474.419,E2 -5474.419} C_VEL
LIN {X 0,Y 512.184,Z 359.301,A -85,B 0,C 180,E1 -5474.687,E2 -5474.687} C_VEL
LIN {X 0,Y 511.615,Z 454.173,A -85,B 0,C 180,E1 -5476.064,E2 -5476.064} C_VEL
LIN {X 0,Y 511.366,Z 467.193,A -85,B 0,C 180,E1 -5476.412,E2 -5476.412} C_VEL
LIN {X 0,Y 511.093,Z 479.254,A -85,B 0,C 180,E1 -5476.886,E2 -5476.886} C_VEL
LIN {X 0,Y 510.833,Z 490.988,A -85,B 0,C 180,E1 -5477.506,E2 -5477.506} C_VEL
LIN {X 0,Y 510.519,Z 502.404,A -85,B 0,C 180,E1 -5478.284,E2 -5478.284} C_VEL
LIN {X 0,Y 510.186,Z 512.965,A -85,B 0,C 180,E1 -5479.182,E2 -5479.182} C_VEL
LIN {X 0,Y 509.885,Z 521.597,A -85,B 0,C 180,E1 -5480.078,E2 -5480.078} C_VEL
LIN {X 0,Y 509.662,Z 529.56,A -85,B 0,C 180,E1 -5481.075,E2 -5481.075} C_VEL
LIN {X 0,Y 509.468,Z 537.338,A -85,B 0,C 180,E1 -5482.27,E2 -5482.27} C_VEL
LIN {X 0,Y 509.308,Z 544.495,A -85,B 0,C 180,E1 -5483.662,E2 -5483.662} C_VEL
LIN {X 0,Y 509.243,Z 549.261,A -85,B 0,C 180,E1 -5484.853,E2 -5484.853} C_VEL
LIN {X 0,Y 509.246,Z 552.904,A -85,B 0,C 180,E1 -5486.043,E2 -5486.043} C_VEL
LIN {X 0,Y 509.2,Z 554.783,A -85,B 0,C 180,E1 -5486.835,E2 -5486.835} C_VEL
LIN {X 0,Y 509.189,Z 556.192,A -85,B 0,C 180,E1 -5487.626,E2 -5487.626} C_VEL
LIN {X 0,Y 509.073,Z 557.811,A -85,B 0,C 180,E1 -5489.209,E2 -5489.209} C_VEL
LIN {X 0,Y 509.069,Z 558.034,A -85,B 0,C 180,E1 -5490,E2 -5490} C_VEL
LIN {X 0,Y 509.112,Z 557.213,A -85,B 0,C 180,E1 -5491.582,E2 -5491.582} C_VEL
LIN {X 0,Y 509.189,Z 556.219,A -85,B 0,C 180,E1 -5492.373,E2 -5492.373} C_VEL
LIN {X 0,Y 509.2,Z 554.817,A -85,B 0,C 180,E1 -5493.164,E2 -5493.164} C_VEL
LIN {X 0,Y 509.204,Z 551.868,A -85,B 0,C 180,E1 -5494.353,E2 -5494.353} C_VEL
LIN {X 0,Y 509.292,Z 547.876,A -85,B 0,C 180,E1 -5495.543,E2 -5495.543} C_VEL
LIN {X 0,Y 509.372,Z 542.183,A -85,B 0,C 180,E1 -5496.844,E2 -5496.844} C_VEL
LIN {X 0,Y 509.543,Z 535.012,A -85,B 0,C 180,E1 -5498.127,E2 -5498.127} C_VEL
LIN {X 0,Y 509.747,Z 526.677,A -85,B 0,C 180,E1 -5499.322,E2 -5499.322} C_VEL
LIN {X 0,Y 509.984,Z 518.116,A -85,B 0,C 180,E1 -5500.32,E2 -5500.32} C_VEL
LIN {X 0,Y 510.379,Z 507.548,A -85,B 0,C 180,E1 -5501.316,E2 -5501.316} C_VEL
LIN {X 0,Y 510.702,Z 495.992,A -85,B 0,C 180,E1 -5502.19,E2 -5502.19} C_VEL
LIN {X 0,Y 510.966,Z 485.58,A -85,B 0,C 180,E1 -5502.814,E2 -5502.814} C_VEL
LIN {X 0,Y 511.241,Z 473.676,A -85,B 0,C 180,E1 -5503.362,E2 -5503.362} C_VEL
LIN {X 0,Y 511.532,Z 459.948,A -85,B 0,C 180,E1 -5503.81,E2 -5503.81} C_VEL
LIN {X 0,Y 511.728,Z 447.553,A -85,B 0,C 180,E1 -5504.058,E2 -5504.058} C_VEL
LIN {X 0,Y 512.098,Z 357.041,A -85,B 0,C 180,E1 -5505.352,E2 -5505.352} C_VEL
LIN {X 0,Y 510.261,Z 345.227,A -85,B 0,C 180,E1 -5505.597,E2 -5505.597} C_VEL
LIN {X 0,Y 510.811,Z 324.508,A -85,B 0,C 180,E1 -5508.864,E2 -5508.864} C_VEL
LIN {X 0,Y 511.317,Z 306.251,A -85,B 0,C 180,E1 -5511.784,E2 -5511.784} C_VEL
LIN {X 0,Y 511.554,Z 295.822,A -85,B 0,C 180,E1 -5513.479,E2 -5513.479} C_VEL
LIN {X 0,Y 509.892,Z 286.971,A -85,B 0,C 180,E1 -5515.057,E2 -5515.057} C_VEL
LIN {X 0,Y 509.897,Z 286.974,A -85,B 0,C 180,E1 -5518.1,E2 -5518.1} C_VEL
LIN {X 0,Y 509.844,Z 286.971,A -85,B 0,C 180,E1 -5521.279,E2 -5521.279} C_VEL
LIN {X 0,Y 509.854,Z 286.979,A -85,B 0,C 180,E1 -5524.202,E2 -5524.202} C_VEL
LIN {X 0,Y 509.814,Z 286.974,A -85,B 0,C 180,E1 -5527.34,E2 -5527.34} C_VEL
LIN {X 0,Y 509.835,Z 286.982,A -85,B 0,C 180,E1 -5530.382,E2 -5530.382} C_VEL
LIN {X 0,Y 509.821,Z 286.975,A -85,B 0,C 180,E1 -5533.062,E2 -5533.062} C_VEL
LIN {X 0,Y 509.827,Z 286.974,A -85,B 0,C 180,E1 -5535.792,E2 -5535.792} C_VEL
LIN {X 0,Y 509.855,Z 286.979,A -85,B 0,C 180,E1 -5538.574,E2 -5538.574} C_VEL
LIN {X 0,Y 509.849,Z 286.97,A -85,B 0,C 180,E1 -5541.786,E2 -5541.786} C_VEL
LIN {X 0,Y 509.838,Z 286.979,A -85,B 0,C 180,E1 -5544.623,E2 -5544.623} C_VEL
LIN {X 0,Y 509.861,Z 286.97,A -85,B 0,C 180,E1 -5547.481,E2 -5547.481} C_VEL
LIN {X 0,Y 509.853,Z 286.971,A -85,B 0,C 180,E1 -5550.273,E2 -5550.273} C_VEL
LIN {X 0,Y 509.88,Z 286.976,A -85,B 0,C 180,E1 -5552.944,E2 -5552.944} C_VEL
LIN {X 0,Y 509.864,Z 286.97,A -85,B 0,C 180,E1 -5555.574,E2 -5555.574} C_VEL
LIN {X 0,Y 509.845,Z 286.978,A -85,B 0,C 180,E1 -5558.998,E2 -5558.998} C_VEL
LIN {X 0,Y 509.883,Z 286.966,A -85,B 0,C 180,E1 -5561.999,E2 -5561.999} C_VEL
LIN {X 0,Y 509.904,Z 286.966,A -85,B 0,C 180,E1 -5564.819,E2 -5564.819} C_VEL
LIN {X 0,Y 509.895,Z 286.965,A -85,B 0,C 180,E1 -5568.124,E2 -5568.124} C_VEL
LIN {X 0,Y 509.91,Z 286.969,A -85,B 0,C 180,E1 -5571.28,E2 -5571.28} C_VEL
LIN {X 0,Y 509.971,Z 286.963,A -85,B 0,C 180,E1 -5573.67,E2 -5573.67} C_VEL
LIN {X 0,Y 510.047,Z 286.955,A -85,B 0,C 180,E1 -5577.631,E2 -5577.631} C_VEL
LIN {X 0,Y 510.048,Z 286.951,A -85,B 0,C 180,E1 -5580,E2 -5580} C_VEL
LIN {X 0,Y 510.047,Z 286.947,A -85,B 0,C 180,E1 -5582.369,E2 -5582.369} C_VEL
LIN {X 0,Y 509.969,Z 286.959,A -85,B 0,C 180,E1 -5585.536,E2 -5585.536} C_VEL
LIN {X 0,Y 509.909,Z 286.963,A -85,B 0,C 180,E1 -5588.721,E2 -5588.721} C_VEL
LIN {X 0,Y 509.899,Z 286.972,A -85,B 0,C 180,E1 -5591.932,E2 -5591.932} C_VEL
LIN {X 0,Y 509.889,Z 286.965,A -85,B 0,C 180,E1 -5595.242,E2 -5595.242} C_VEL
LIN {X 0,Y 509.855,Z 286.975,A -85,B 0,C 180,E1 -5598.484,E2 -5598.484} C_VEL
LIN {X 0,Y 509.845,Z 286.971,A -85,B 0,C 180,E1 -5601.002,E2 -5601.002} C_VEL
LIN {X 0,Y 509.817,Z 286.974,A -85,B 0,C 180,E1 -5603.564,E2 -5603.564} C_VEL
LIN {X 0,Y 509.88,Z 286.975,A -85,B 0,C 180,E1 -5606.373,E2 -5606.373} C_VEL
LIN {X 0,Y 509.853,Z 286.97,A -85,B 0,C 180,E1 -5609.752,E2 -5609.752} C_VEL
LIN {X 0,Y 509.869,Z 286.975,A -85,B 0,C 180,E1 -5612.775,E2 -5612.775} C_VEL
LIN {X 0,Y 509.822,Z 286.973,A -85,B 0,C 180,E1 -5615.579,E2 -5615.579} C_VEL
LIN {X 0,Y 509.846,Z 286.974,A -85,B 0,C 180,E1 -5618.339,E2 -5618.339} C_VEL
LIN {X 0,Y 509.847,Z 286.972,A -85,B 0,C 180,E1 -5621.427,E2 -5621.427} C_VEL
LIN {X 0,Y 509.837,Z 286.977,A -85,B 0,C 180,E1 -5624.671,E2 -5624.671} C_VEL
LIN {X 0,Y 509.803,Z 286.978,A -85,B 0,C 180,E1 -5627.508,E2 -5627.508} C_VEL
LIN {X 0,Y 509.831,Z 286.975,A -85,B 0,C 180,E1 -5630.647,E2 -5630.647} C_VEL
LIN {X 0,Y 509.806,Z 286.978,A -85,B 0,C 180,E1 -5633.718,E2 -5633.718} C_VEL
LIN {X 0,Y 509.146,Z 287.058,A -85,B 0,C 180,E1 -5634.378,E2 -5634.378} C_VEL
LIN {X 0,Y 506.341,Z 287.413,A -85,B 0,C 180,E1 -5635.45,E2 -5635.45} C_VEL
LIN {X 0,Y 503.956,Z 287.712,A -85,B 0,C 180,E1 -5636.314,E2 -5636.314} C_VEL
LIN {X 0,Y 502.906,Z 287.84,A -85,B 0,C 180,E1 -5636.98,E2 -5636.98} C_VEL
LIN {X 0,Y 502.807,Z 287.85,A -85,B 0,C 180,E1 -5637.205,E2 -5637.205} C_VEL
LIN {X 0,Y 502.81,Z 287.848,A -85,B 0,C 180,E1 -5640.067,E2 -5640.067} C_VEL
LIN {X 0,Y 502.783,Z 287.86,A -85,B 0,C 180,E1 -5643.43,E2 -5643.43} C_VEL
LIN {X 0,Y 502.767,Z 287.854,A -85,B 0,C 180,E1 -5646.086,E2 -5646.086} C_VEL
LIN {X 0,Y 502.783,Z 287.85,A -85,B 0,C 180,E1 -5648.689,E2 -5648.689} C_VEL
LIN {X 0,Y 502.805,Z 287.851,A -85,B 0,C 180,E1 -5651.248,E2 -5651.248} C_VEL
LIN {X 0,Y 502.852,Z 287.842,A -85,B 0,C 180,E1 -5654.601,E2 -5654.601} C_VEL
LIN {X 0,Y 502.873,Z 287.845,A -85,B 0,C 180,E1 -5658.044,E2 -5658.044} C_VEL
LIN {X 0,Y 502.84,Z 287.844,A -85,B 0,C 180,E1 -5661.157,E2 -5661.157} C_VEL
LIN {X 0,Y 502.872,Z 287.843,A -85,B 0,C 180,E1 -5663.581,E2 -5663.581} C_VEL
LIN {X 0,Y 502.743,Z 287.864,A -85,B 0,C 180,E1 -5665.992,E2 -5665.992} C_VEL
LIN {X 0,Y 503.006,Z 287.825,A -85,B 0,C 180,E1 -5667.598,E2 -5667.598} C_VEL
LIN {X 0,Y 503.006,Z 287.829,A -85,B 0,C 180,E1 -5670,E2 -5670} C_VEL
LIN {X 0,Y 503.004,Z 287.83,A -85,B 0,C 180,E1 -5672.403,E2 -5672.403} C_VEL
LIN {X 0,Y 502.894,Z 287.837,A -85,B 0,C 180,E1 -5675.614,E2 -5675.614} C_VEL
LIN {X 0,Y 502.85,Z 287.846,A -85,B 0,C 180,E1 -5678.035,E2 -5678.035} C_VEL
LIN {X 0,Y 502.833,Z 287.844,A -85,B 0,C 180,E1 -5681.285,E2 -5681.285} C_VEL
LIN {X 0,Y 502.799,Z 287.858,A -85,B 0,C 180,E1 -5684.573,E2 -5684.573} C_VEL
LIN {X 0,Y 502.789,Z 287.85,A -85,B 0,C 180,E1 -5687.91,E2 -5687.91} C_VEL
LIN {X 0,Y 502.807,Z 287.854,A -85,B 0,C 180,E1 -5690.528,E2 -5690.528} C_VEL
LIN {X 0,Y 502.785,Z 287.858,A -85,B 0,C 180,E1 -5693.041,E2 -5693.041} C_VEL
LIN {X 0,Y 502.759,Z 287.858,A -85,B 0,C 180,E1 -5695.68,E2 -5695.68} C_VEL
LIN {X 0,Y 502.796,Z 287.927,A -85,B 0,C 180,E1 -5696.85,E2 -5696.85} C_VEL
LIN {X 0,Y 503.607,Z 293.952,A -85,B 0,C 180,E1 -5698.099,E2 -5698.099} C_VEL
LIN {X 0,Y 503.262,Z 309.179,A -85,B 0,C 180,E1 -5701.112,E2 -5701.112} C_VEL
LIN {X 0,Y 503.244,Z 309.907,A -85,B 0,C 180,E1 -5701.254,E2 -5701.254} C_VEL
LIN {X 0,Y 505.44,Z 322.215,A -85,B 0,C 180,E1 -5701.516,E2 -5701.516} C_VEL
LIN {X 0,Y 504.854,Z 417.36,A -85,B 0,C 180,E1 -5702.921,E2 -5702.921} C_VEL
LIN {X 0,Y 504.582,Z 430.938,A -85,B 0,C 180,E1 -5703.294,E2 -5703.294} C_VEL
LIN {X 0,Y 504.308,Z 443.333,A -85,B 0,C 180,E1 -5703.8,E2 -5703.8} C_VEL
LIN {X 0,Y 503.962,Z 455.373,A -85,B 0,C 180,E1 -5704.467,E2 -5704.467} C_VEL
LIN {X 0,Y 503.672,Z 466.543,A -85,B 0,C 180,E1 -5705.263,E2 -5705.263} C_VEL
LIN {X 0,Y 503.342,Z 476.584,A -85,B 0,C 180,E1 -5706.151,E2 -5706.151} C_VEL
LIN {X 0,Y 502.962,Z 486.183,A -85,B 0,C 180,E1 -5707.205,E2 -5707.205} C_VEL
LIN {X 0,Y 502.719,Z 493.719,A -85,B 0,C 180,E1 -5708.212,E2 -5708.212} C_VEL
LIN {X 0,Y 502.492,Z 500.734,A -85,B 0,C 180,E1 -5709.353,E2 -5709.353} C_VEL
LIN {X 0,Y 502.323,Z 506.434,A -85,B 0,C 180,E1 -5710.493,E2 -5710.493} C_VEL
LIN {X 0,Y 502.23,Z 510.981,A -85,B 0,C 180,E1 -5711.623,E2 -5711.623} C_VEL
LIN {X 0,Y 502.167,Z 514.533,A -85,B 0,C 180,E1 -5712.745,E2 -5712.745} C_VEL
LIN {X 0,Y 502.092,Z 517.185,A -85,B 0,C 180,E1 -5713.858,E2 -5713.858} C_VEL
LIN {X 0,Y 502.077,Z 518.269,A -85,B 0,C 180,E1 -5714.447,E2 -5714.447} C_VEL
LIN {X 0,Y 502.016,Z 519.675,A -85,B 0,C 180,E1 -5715.574,E2 -5715.574} C_VEL
LIN {X 0,Y 501.996,Z 520.311,A -85,B 0,C 180,E1 -5716.72,E2 -5716.72} C_VEL
LIN {X 0,Y 501.998,Z 520.13,A -85,B 0,C 180,E1 -5717.903,E2 -5717.903} C_VEL
LIN {X 0,Y 502.019,Z 519.056,A -85,B 0,C 180,E1 -5719.111,E2 -5719.111} C_VEL
LIN {X 0,Y 502.063,Z 517.006,A -85,B 0,C 180,E1 -5720.345,E2 -5720.345} C_VEL
LIN {X 0,Y 502.184,Z 513.881,A -85,B 0,C 180,E1 -5721.602,E2 -5721.602} C_VEL
LIN {X 0,Y 502.308,Z 509.005,A -85,B 0,C 180,E1 -5723.013,E2 -5723.013} C_VEL
LIN {X 0,Y 502.47,Z 502.547,A -85,B 0,C 180,E1 -5724.424,E2 -5724.424} C_VEL
LIN {X 0,Y 502.666,Z 495.816,A -85,B 0,C 180,E1 -5725.579,E2 -5725.579} C_VEL
LIN {X 0,Y 502.985,Z 487.447,A -85,B 0,C 180,E1 -5726.741,E2 -5726.741} C_VEL
LIN {X 0,Y 503.3,Z 477.746,A -85,B 0,C 180,E1 -5727.834,E2 -5727.834} C_VEL
LIN {X 0,Y 503.577,Z 467.922,A -85,B 0,C 180,E1 -5728.73,E2 -5728.73} C_VEL
LIN {X 0,Y 503.975,Z 456.405,A -85,B 0,C 180,E1 -5729.564,E2 -5729.564} C_VEL
LIN {X 0,Y 504.275,Z 444.655,A -85,B 0,C 180,E1 -5730.231,E2 -5730.231} C_VEL
LIN {X 0,Y 504.536,Z 432.033,A -85,B 0,C 180,E1 -5730.764,E2 -5730.764} C_VEL
LIN {X 0,Y 504.767,Z 419.258,A -85,B 0,C 180,E1 -5731.128,E2 -5731.128} C_VEL
LIN {X 0,Y 504.916,Z 396.494,A -85,B 0,C 180,E1 -5731.495,E2 -5731.495} C_VEL
LIN {X 0,Y 505.374,Z 321.16,A -85,B 0,C 180,E1 -5732.598,E2 -5732.598} C_VEL
LIN {X 0,Y 503.245,Z 309.22,A -85,B 0,C 180,E1 -5732.867,E2 -5732.867} C_VEL
LIN {X 0,Y 503.269,Z 291.237,A -85,B 0,C 180,E1 -5735.891,E2 -5735.891} C_VEL
LIN {X 0,Y 502.883,Z 287.846,A -85,B 0,C 180,E1 -5736.473,E2 -5736.473} C_VEL
LIN {X 0,Y 502.838,Z 287.852,A -85,B 0,C 180,E1 -5739.548,E2 -5739.548} C_VEL
LIN {X 0,Y 502.825,Z 287.85,A -85,B 0,C 180,E1 -5742.091,E2 -5742.091} C_VEL
LIN {X 0,Y 502.854,Z 287.852,A -85,B 0,C 180,E1 -5745.429,E2 -5745.429} C_VEL
LIN {X 0,Y 502.879,Z 287.84,A -85,B 0,C 180,E1 -5748.717,E2 -5748.717} C_VEL
LIN {X 0,Y 502.902,Z 287.842,A -85,B 0,C 180,E1 -5751.966,E2 -5751.966} C_VEL
LIN {X 0,Y 502.933,Z 287.835,A -85,B 0,C 180,E1 -5754.386,E2 -5754.386} C_VEL
LIN {X 0,Y 503.025,Z 287.827,A -85,B 0,C 180,E1 -5757.598,E2 -5757.598} C_VEL
LIN {X 0,Y 503.029,Z 287.828,A -85,B 0,C 180,E1 -5760,E2 -5760} C_VEL
LIN {X 0,Y 503.026,Z 287.824,A -85,B 0,C 180,E1 -5762.402,E2 -5762.402} C_VEL
LIN {X 0,Y 502.927,Z 287.836,A -85,B 0,C 180,E1 -5765.613,E2 -5765.613} C_VEL
LIN {X 0,Y 502.871,Z 287.841,A -85,B 0,C 180,E1 -5768.843,E2 -5768.843} C_VEL
LIN {X 0,Y 502.848,Z 287.849,A -85,B 0,C 180,E1 -5772.101,E2 -5772.101} C_VEL
LIN {X 0,Y 502.85,Z 287.843,A -85,B 0,C 180,E1 -5775.4,E2 -5775.4} C_VEL
LIN {X 0,Y 502.828,Z 287.852,A -85,B 0,C 180,E1 -5778.752,E2 -5778.752} C_VEL
LIN {X 0,Y 502.784,Z 287.85,A -85,B 0,C 180,E1 -5781.311,E2 -5781.311} C_VEL
LIN {X 0,Y 502.786,Z 287.85,A -85,B 0,C 180,E1 -5783.914,E2 -5783.914} C_VEL
LIN {X 0,Y 502.866,Z 287.846,A -85,B 0,C 180,E1 -5786.566,E2 -5786.566} C_VEL
LIN {X 0,Y 502.825,Z 287.849,A -85,B 0,C 180,E1 -5789.288,E2 -5789.288} C_VEL
LIN {X 0,Y 502.784,Z 287.85,A -85,B 0,C 180,E1 -5792.085,E2 -5792.085} C_VEL
LIN {X 0,Y 502.796,Z 287.855,A -85,B 0,C 180,E1 -5794.966,E2 -5794.966} C_VEL
LIN {X 0,Y 502.794,Z 287.849,A -85,B 0,C 180,E1 -5797.954,E2 -5797.954} C_VEL
LIN {X 0,Y 502.821,Z 287.852,A -85,B 0,C 180,E1 -5801.066,E2 -5801.066} C_VEL
LIN {X 0,Y 502.787,Z 287.852,A -85,B 0,C 180,E1 -5804.53,E2 -5804.53} C_VEL
LIN {X 0,Y 502.797,Z 287.853,A -85,B 0,C 180,E1 -5807.86,E2 -5807.86} C_VEL
LIN {X 0,Y 502.803,Z 287.851,A -85,B 0,C 180,E1 -5811.024,E2 -5811.024} C_VEL
LIN {X 0,Y 502.777,Z 287.858,A -85,B 0,C 180,E1 -5814.169,E2 -5814.169} C_VEL
LIN {X 0,Y 502.835,Z 287.849,A -85,B 0,C 180,E1 -5816.993,E2 -5816.993} C_VEL
LIN {X 0,Y 502.818,Z 287.854,A -85,B 0,C 180,E1 -5820.065,E2 -5820.065} C_VEL
LIN {X 0,Y 502.833,Z 287.851,A -85,B 0,C 180,E1 -5822.533,E2 -5822.533} C_VEL
LIN {X 0,Y 502.875,Z 287.98,A -85,B 0,C 180,E1 -5825.211,E2 -5825.211} C_VEL
LIN {X 0,Y 504.306,Z 296.104,A -85,B 0,C 180,E1 -5826.579,E2 -5826.579} C_VEL
LIN {X 0,Y 504.044,Z 309.788,A -85,B 0,C 180,E1 -5828.744,E2 -5828.744} C_VEL
LIN {X 0,Y 503.592,Z 329.695,A -85,B 0,C 180,E1 -5831.868,E2 -5831.868} C_VEL
LIN {X 0,Y 503.229,Z 344.621,A -85,B 0,C 180,E1 -5834.193,E2 -5834.193} C_VEL
LIN {X 0,Y 505.324,Z 359.069,A -85,B 0,C 180,E1 -5834.474,E2 -5834.474} C_VEL
LIN {X 0,Y 504.728,Z 453.615,A -85,B 0,C 180,E1 -5835.87,E2 -5835.87} C_VEL
LIN {X 0,Y 504.451,Z 467.484,A -85,B 0,C 180,E1 -5836.248,E2 -5836.248} C_VEL
LIN {X 0,Y 504.117,Z 479.942,A -85,B 0,C 180,E1 -5836.752,E2 -5836.752} C_VEL
LIN {X 0,Y 503.825,Z 492.316,A -85,B 0,C 180,E1 -5837.439,E2 -5837.439} C_VEL
LIN {X 0,Y 503.503,Z 503.346,A -85,B 0,C 180,E1 -5838.221,E2 -5838.221} C_VEL
LIN {X 0,Y 503.148,Z 513.693,A -85,B 0,C 180,E1 -5839.13,E2 -5839.13} C_VEL
LIN {X 0,Y 502.81,Z 522.98,A -85,B 0,C 180,E1 -5840.141,E2 -5840.141} C_VEL
LIN {X 0,Y 502.533,Z 532.016,A -85,B 0,C 180,E1 -5841.353,E2 -5841.353} C_VEL
LIN {X 0,Y 502.346,Z 539.295,A -85,B 0,C 180,E1 -5842.564,E2 -5842.564} C_VEL
LIN {X 0,Y 502.235,Z 544.205,A -85,B 0,C 180,E1 -5843.572,E2 -5843.572} C_VEL
LIN {X 0,Y 502.174,Z 548.979,A -85,B 0,C 180,E1 -5844.78,E2 -5844.78} C_VEL
LIN {X 0,Y 502.139,Z 552.627,A -85,B 0,C 180,E1 -5845.987,E2 -5845.987} C_VEL
LIN {X 0,Y 502.12,Z 554.511,A -85,B 0,C 180,E1 -5846.79,E2 -5846.79} C_VEL
LIN {X 0,Y 502.091,Z 555.922,A -85,B 0,C 180,E1 -5847.593,E2 -5847.593} C_VEL
LIN {X 0,Y 501.99,Z 557.547,A -85,B 0,C 180,E1 -5849.197,E2 -5849.197} C_VEL
LIN {X 0,Y 501.983,Z 557.77,A -85,B 0,C 180,E1 -5850,E2 -5850} C_VEL
LIN {X 0,Y 502.036,Z 556.951,A -85,B 0,C 180,E1 -5851.604,E2 -5851.604} C_VEL
LIN {X 0,Y 502.091,Z 555.955,A -85,B 0,C 180,E1 -5852.406,E2 -5852.406} C_VEL
LIN {X 0,Y 502.12,Z 554.552,A -85,B 0,C 180,E1 -5853.209,E2 -5853.209} C_VEL
LIN {X 0,Y 502.102,Z 551.6,A -85,B 0,C 180,E1 -5854.415,E2 -5854.415} C_VEL
LIN {X 0,Y 502.208,Z 547.605,A -85,B 0,C 180,E1 -5855.621,E2 -5855.621} C_VEL
LIN {X 0,Y 502.323,Z 541.552,A -85,B 0,C 180,E1 -5857.011,E2 -5857.011} C_VEL
LIN {X 0,Y 502.475,Z 534.726,A -85,B 0,C 180,E1 -5858.242,E2 -5858.242} C_VEL
LIN {X 0,Y 502.712,Z 526.384,A -85,B 0,C 180,E1 -5859.454,E2 -5859.454} C_VEL
LIN {X 0,Y 502.965,Z 517.81,A -85,B 0,C 180,E1 -5860.465,E2 -5860.465} C_VEL
LIN {X 0,Y 503.398,Z 507.23,A -85,B 0,C 180,E1 -5861.475,E2 -5861.475} C_VEL
LIN {X 0,Y 503.738,Z 495.658,A -85,B 0,C 180,E1 -5862.362,E2 -5862.362} C_VEL
LIN {X 0,Y 504.026,Z 485.223,A -85,B 0,C 180,E1 -5862.993,E2 -5862.993} C_VEL
LIN {X 0,Y 504.33,Z 473.283,A -85,B 0,C 180,E1 -5863.549,E2 -5863.549} C_VEL
LIN {X 0,Y 504.624,Z 460.417,A -85,B 0,C 180,E1 -5863.977,E2 -5863.977} C_VEL
LIN {X 0,Y 504.856,Z 446.946,A -85,B 0,C 180,E1 -5864.254,E2 -5864.254} C_VEL
LIN {X 0,Y 505.194,Z 357.592,A -85,B 0,C 180,E1 -5865.555,E2 -5865.555} C_VEL
LIN {X 0,Y 503.257,Z 344.95,A -85,B 0,C 180,E1 -5865.824,E2 -5865.824} C_VEL
LIN {X 0,Y 503.813,Z 325.572,A -85,B 0,C 180,E1 -5868.924,E2 -5868.924} C_VEL
LIN {X 0,Y 504.367,Z 307.339,A -85,B 0,C 180,E1 -5871.884,E2 -5871.884} C_VEL
LIN {X 0,Y 504.672,Z 297.815,A -85,B 0,C 180,E1 -5873.45,E2 -5873.45} C_VEL
LIN {X 0,Y 502.855,Z 287.849,A -85,B 0,C 180,E1 -5875.23,E2 -5875.23} C_VEL
LIN {X 0,Y 502.843,Z 287.85,A -85,B 0,C 180,E1 -5878.295,E2 -5878.295} C_VEL
LIN {X 0,Y 502.791,Z 287.851,A -85,B 0,C 180,E1 -5881.498,E2 -5881.498} C_VEL
LIN {X 0,Y 502.802,Z 287.854,A -85,B 0,C 180,E1 -5883.993,E2 -5883.993} C_VEL
LIN {X 0,Y 502.775,Z 287.851,A -85,B 0,C 180,E1 -5887.177,E2 -5887.177} C_VEL
LIN {X 0,Y 502.785,Z 287.854,A -85,B 0,C 180,E1 -5890.015,E2 -5890.015} C_VEL
LIN {X 0,Y 502.799,Z 287.854,A -85,B 0,C 180,E1 -5892.199,E2 -5892.199} C_VEL
LIN {X 0,Y 502.797,Z 287.849,A -85,B 0,C 180,E1 -5895.468,E2 -5895.468} C_VEL
LIN {X 0,Y 502.826,Z 287.846,A -85,B 0,C 180,E1 -5897.864,E2 -5897.864} C_VEL
LIN {X 0,Y 502.799,Z 287.852,A -85,B 0,C 180,E1 -5901.024,E2 -5901.024} C_VEL
LIN {X 0,Y 502.778,Z 287.853,A -85,B 0,C 180,E1 -5904.167,E2 -5904.167} C_VEL
LIN {X 0,Y 502.828,Z 287.852,A -85,B 0,C 180,E1 -5906.993,E2 -5906.993} C_VEL
LIN {X 0,Y 502.81,Z 287.847,A -85,B 0,C 180,E1 -5910.064,E2 -5910.064} C_VEL
LIN {X 0,Y 502.828,Z 287.848,A -85,B 0,C 180,E1 -5912.533,E2 -5912.533} C_VEL
LIN {X 0,Y 502.823,Z 287.851,A -85,B 0,C 180,E1 -5915.298,E2 -5915.298} C_VEL
LIN {X 0,Y 502.775,Z 287.852,A -85,B 0,C 180,E1 -5917.826,E2 -5917.826} C_VEL
LIN {X 0,Y 502.819,Z 287.846,A -85,B 0,C 180,E1 -5920.4,E2 -5920.4} C_VEL
LIN {X 0,Y 502.828,Z 287.849,A -85,B 0,C 180,E1 -5922.932,E2 -5922.932} C_VEL
LIN {X 0,Y 502.846,Z 287.851,A -85,B 0,C 180,E1 -5925.429,E2 -5925.429} C_VEL
LIN {X 0,Y 502.871,Z 287.84,A -85,B 0,C 180,E1 -5928.717,E2 -5928.717} C_VEL
LIN {X 0,Y 502.896,Z 287.839,A -85,B 0,C 180,E1 -5931.967,E2 -5931.967} C_VEL
LIN {X 0,Y 502.932,Z 287.832,A -85,B 0,C 180,E1 -5934.387,E2 -5934.387} C_VEL
LIN {X 0,Y 503.017,Z 287.83,A -85,B 0,C 180,E1 -5937.598,E2 -5937.598} C_VEL
LIN {X 0,Y 503.02,Z 287.826,A -85,B 0,C 180,E1 -5940,E2 -5940} C_VEL
LIN {X 0,Y 503.017,Z 287.823,A -85,B 0,C 180,E1 -5942.402,E2 -5942.402} C_VEL
LIN {X 0,Y 502.922,Z 287.838,A -85,B 0,C 180,E1 -5945.614,E2 -5945.614} C_VEL
LIN {X 0,Y 502.867,Z 287.84,A -85,B 0,C 180,E1 -5948.844,E2 -5948.844} C_VEL
LIN {X 0,Y 502.84,Z 287.852,A -85,B 0,C 180,E1 -5952.102,E2 -5952.102} C_VEL
LIN {X 0,Y 502.843,Z 287.843,A -85,B 0,C 180,E1 -5955.4,E2 -5955.4} C_VEL
LIN {X 0,Y 502.82,Z 287.848,A -85,B 0,C 180,E1 -5958.752,E2 -5958.752} C_VEL
LIN {X 0,Y 502.778,Z 287.851,A -85,B 0,C 180,E1 -5961.312,E2 -5961.312} C_VEL
LIN {X 0,Y 502.769,Z 287.855,A -85,B 0,C 180,E1 -5963.915,E2 -5963.915} C_VEL
LIN {X 0,Y 502.831,Z 287.852,A -85,B 0,C 180,E1 -5966.568,E2 -5966.568} C_VEL
LIN {X 0,Y 502.811,Z 287.848,A -85,B 0,C 180,E1 -5969.936,E2 -5969.936} C_VEL
LIN {X 0,Y 502.828,Z 287.848,A -85,B 0,C 180,E1 -5973.032,E2 -5973.032} C_VEL
LIN {X 0,Y 502.77,Z 287.853,A -85,B 0,C 180,E1 -5975.952,E2 -5975.952} C_VEL
LIN {X 0,Y 502.791,Z 287.856,A -85,B 0,C 180,E1 -5978.978,E2 -5978.978} C_VEL
LIN {X 0,Y 502.801,Z 287.849,A -85,B 0,C 180,E1 -5982.2,E2 -5982.2} C_VEL
LIN {X 0,Y 502.784,Z 287.853,A -85,B 0,C 180,E1 -5985.471,E2 -5985.471} C_VEL
LIN {X 0,Y 502.793,Z 287.849,A -85,B 0,C 180,E1 -5987.861,E2 -5987.861} C_VEL
LIN {X 0,Y 502.792,Z 287.858,A -85,B 0,C 180,E1 -5991.024,E2 -5991.024} C_VEL
LIN {X 0,Y 502.771,Z 287.852,A -85,B 0,C 180,E1 -5994.171,E2 -5994.171} C_VEL
LIN {X 0,Y 502.807,Z 287.85,A -85,B 0,C 180,E1 -5997.205,E2 -5997.205} C_VEL
LIN {X 0,Y 502.104,Z 287.937,A -85,B 0,C 180,E1 -5997.874,E2 -5997.874} C_VEL
LIN {X 0,Y 499.243,Z 288.295,A -85,B 0,C 180,E1 -5998.96,E2 -5998.96} C_VEL
LIN {X 0,Y 496.843,Z 288.593,A -85,B 0,C 180,E1 -5999.835,E2 -5999.835} C_VEL
LIN {X 0,Y 495.812,Z 288.719,A -85,B 0,C 180,E1 -6000.51,E2 -6000.51} C_VEL
LIN {X 0,Y 495.726,Z 288.731,A -85,B 0,C 180,E1 -6000.739,E2 -6000.739} C_VEL
LIN {X 0,Y 495.713,Z 288.734,A -85,B 0,C 180,E1 -6003.928,E2 -6003.928} C_VEL
LIN {X 0,Y 495.761,Z 288.729,A -85,B 0,C 180,E1 -6007.141,E2 -6007.141} C_VEL
LIN {X 0,Y 495.759,Z 288.728,A -85,B 0,C 180,E1 -6010.11,E2 -6010.11} C_VEL
LIN {X 0,Y 495.74,Z 288.728,A -85,B 0,C 180,E1 -6012.68,E2 -6012.68} C_VEL
LIN {X 0,Y 495.791,Z 288.723,A -85,B 0,C 180,E1 -6015.218,E2 -6015.218} C_VEL
LIN {X 0,Y 495.824,Z 288.718,A -85,B 0,C 180,E1 -6018.555,E2 -6018.555} C_VEL
LIN {X 0,Y 495.814,Z 288.727,A -85,B 0,C 180,E1 -6021.852,E2 -6021.852} C_VEL
LIN {X 0,Y 495.854,Z 288.718,A -85,B 0,C 180,E1 -6024.307,E2 -6024.307} C_VEL
LIN {X 0,Y 495.972,Z 288.701,A -85,B 0,C 180,E1 -6027.564,E2 -6027.564} C_VEL
LIN {X 0,Y 495.975,Z 288.705,A -85,B 0,C 180,E1 -6030,E2 -6030} C_VEL
LIN {X 0,Y 495.97,Z 288.705,A -85,B 0,C 180,E1 -6032.437,E2 -6032.437} C_VEL
LIN {X 0,Y 495.853,Z 288.715,A -85,B 0,C 180,E1 -6035.694,E2 -6035.694} C_VEL
LIN {X 0,Y 495.814,Z 288.724,A -85,B 0,C 180,E1 -6038.149,E2 -6038.149} C_VEL
LIN {X 0,Y 495.792,Z 288.721,A -85,B 0,C 180,E1 -6041.447,E2 -6041.447} C_VEL
LIN {X 0,Y 495.748,Z 288.733,A -85,B 0,C 180,E1 -6044.785,E2 -6044.785} C_VEL
LIN {X 0,Y 495.766,Z 288.727,A -85,B 0,C 180,E1 -6048.173,E2 -6048.173} C_VEL
LIN {X 0,Y 495.769,Z 288.734,A -85,B 0,C 180,E1 -6050.757,E2 -6050.757} C_VEL
LIN {X 0,Y 495.734,Z 288.733,A -85,B 0,C 180,E1 -6053.388,E2 -6053.388} C_VEL
LIN {X 0,Y 495.755,Z 288.755,A -85,B 0,C 180,E1 -6056.693,E2 -6056.693} C_VEL
LIN {X 0,Y 496.619,Z 294.192,A -85,B 0,C 180,E1 -6057.84,E2 -6057.84} C_VEL
LIN {X 0,Y 496.293,Z 309.396,A -85,B 0,C 180,E1 -6060.887,E2 -6060.887} C_VEL
LIN {X 0,Y 496.271,Z 310.183,A -85,B 0,C 180,E1 -6061.036,E2 -6061.036} C_VEL
LIN {X 0,Y 498.547,Z 322.071,A -85,B 0,C 180,E1 -6061.291,E2 -6061.291} C_VEL
LIN {X 0,Y 497.959,Z 417.815,A -85,B 0,C 180,E1 -6062.733,E2 -6062.733} C_VEL
LIN {X 0,Y 497.674,Z 431.481,A -85,B 0,C 180,E1 -6063.116,E2 -6063.116} C_VEL
LIN {X 0,Y 497.411,Z 443.511,A -85,B 0,C 180,E1 -6063.615,E2 -6063.615} C_VEL
LIN {X 0,Y 497.009,Z 456.094,A -85,B 0,C 180,E1 -6064.325,E2 -6064.325} C_VEL
LIN {X 0,Y 496.702,Z 466.683,A -85,B 0,C 180,E1 -6065.092,E2 -6065.092} C_VEL
LIN {X 0,Y 496.375,Z 476.445,A -85,B 0,C 180,E1 -6065.964,E2 -6065.964} C_VEL
LIN {X 0,Y 495.98,Z 486.122,A -85,B 0,C 180,E1 -6067.029,E2 -6067.029} C_VEL
LIN {X 0,Y 495.68,Z 493.914,A -85,B 0,C 180,E1 -6068.081,E2 -6068.081} C_VEL
LIN {X 0,Y 495.48,Z 500.594,A -85,B 0,C 180,E1 -6069.173,E2 -6069.173} C_VEL
LIN {X 0,Y 495.282,Z 506.415,A -85,B 0,C 180,E1 -6070.338,E2 -6070.338} C_VEL
LIN {X 0,Y 495.173,Z 511.089,A -85,B 0,C 180,E1 -6071.503,E2 -6071.503} C_VEL
LIN {X 0,Y 495.06,Z 515.505,A -85,B 0,C 180,E1 -6072.955,E2 -6072.955} C_VEL
LIN {X 0,Y 495.006,Z 517.946,A -85,B 0,C 180,E1 -6074.083,E2 -6074.083} C_VEL
LIN {X 0,Y 494.942,Z 519.622,A -85,B 0,C 180,E1 -6075.234,E2 -6075.234} C_VEL
LIN {X 0,Y 494.898,Z 520.499,A -85,B 0,C 180,E1 -6076.406,E2 -6076.406} C_VEL
LIN {X 0,Y 494.919,Z 520.538,A -85,B 0,C 180,E1 -6077.597,E2 -6077.597} C_VEL
LIN {X 0,Y 494.927,Z 519.218,A -85,B 0,C 180,E1 -6079.216,E2 -6079.216} C_VEL
LIN {X 0,Y 495.018,Z 516.345,A -85,B 0,C 180,E1 -6080.818,E2 -6080.818} C_VEL
LIN {X 0,Y 495.16,Z 511.864,A -85,B 0,C 180,E1 -6082.387,E2 -6082.387} C_VEL
LIN {X 0,Y 495.322,Z 506.606,A -85,B 0,C 180,E1 -6083.73,E2 -6083.73} C_VEL
LIN {X 0,Y 495.493,Z 500.678,A -85,B 0,C 180,E1 -6084.922,E2 -6084.922} C_VEL
LIN {X 0,Y 495.76,Z 492.817,A -85,B 0,C 180,E1 -6086.191,E2 -6086.191} C_VEL
LIN {X 0,Y 496.071,Z 484.133,A -85,B 0,C 180,E1 -6087.313,E2 -6087.313} C_VEL
LIN {X 0,Y 496.425,Z 473.646,A -85,B 0,C 180,E1 -6088.411,E2 -6088.411} C_VEL
LIN {X 0,Y 496.808,Z 463.435,A -85,B 0,C 180,E1 -6089.267,E2 -6089.267} C_VEL
LIN {X 0,Y 497.191,Z 452.383,A -85,B 0,C 180,E1 -6090.004,E2 -6090.004} C_VEL
LIN {X 0,Y 497.516,Z 441.172,A -85,B 0,C 180,E1 -6090.59,E2 -6090.59} C_VEL
LIN {X 0,Y 497.726,Z 428.456,A -85,B 0,C 180,E1 -6091.083,E2 -6091.083} C_VEL
LIN {X 0,Y 497.947,Z 415.461,A -85,B 0,C 180,E1 -6091.409,E2 -6091.409} C_VEL
LIN {X 0,Y 498.508,Z 321.637,A -85,B 0,C 180,E1 -6092.816,E2 -6092.816} C_VEL
LIN {X 0,Y 496.264,Z 309.415,A -85,B 0,C 180,E1 -6093.103,E2 -6093.103} C_VEL
LIN {X 0,Y 496.324,Z 292.398,A -85,B 0,C 180,E1 -6095.977,E2 -6095.977} C_VEL
LIN {X 0,Y 495.828,Z 288.725,A -85,B 0,C 180,E1 -6096.616,E2 -6096.616} C_VEL
LIN {X 0,Y 495.773,Z 288.727,A -85,B 0,C 180,E1 -6100.109,E2 -6100.109} C_VEL
LIN {X 0,Y 495.767,Z 288.73,A -85,B 0,C 180,E1 -6102.68,E2 -6102.68} C_VEL
LIN {X 0,Y 495.797,Z 288.731,A -85,B 0,C 180,E1 -6105.217,E2 -6105.217} C_VEL
LIN {X 0,Y 495.853,Z 288.715,A -85,B 0,C 180,E1 -6108.555,E2 -6108.555} C_VEL
LIN {X 0,Y 495.873,Z 288.72,A -85,B 0,C 180,E1 -6111.852,E2 -6111.852} C_VEL
LIN {X 0,Y 495.889,Z 288.713,A -85,B 0,C 180,E1 -6114.306,E2 -6114.306} C_VEL
LIN {X 0,Y 495.994,Z 288.703,A -85,B 0,C 180,E1 -6117.563,E2 -6117.563} C_VEL
LIN {X 0,Y 495.984,Z 288.697,A -85,B 0,C 180,E1 -6120.812,E2 -6120.812} C_VEL
LIN {X 0,Y 495.995,Z 288.7,A -85,B 0,C 180,E1 -6122.436,E2 -6122.436} C_VEL
LIN {X 0,Y 495.882,Z 288.714,A -85,B 0,C 180,E1 -6125.693,E2 -6125.693} C_VEL
LIN {X 0,Y 495.84,Z 288.716,A -85,B 0,C 180,E1 -6128.97,E2 -6128.97} C_VEL
LIN {X 0,Y 495.812,Z 288.728,A -85,B 0,C 180,E1 -6132.276,E2 -6132.276} C_VEL
LIN {X 0,Y 495.825,Z 288.718,A -85,B 0,C 180,E1 -6135.451,E2 -6135.451} C_VEL
LIN {X 0,Y 495.78,Z 288.726,A -85,B 0,C 180,E1 -6138.237,E2 -6138.237} C_VEL
LIN {X 0,Y 495.776,Z 288.728,A -85,B 0,C 180,E1 -6140.756,E2 -6140.756} C_VEL
LIN {X 0,Y 495.749,Z 288.727,A -85,B 0,C 180,E1 -6143.387,E2 -6143.387} C_VEL
LIN {X 0,Y 495.792,Z 288.722,A -85,B 0,C 180,E1 -6146.068,E2 -6146.068} C_VEL
LIN {X 0,Y 495.774,Z 288.729,A -85,B 0,C 180,E1 -6148.815,E2 -6148.815} C_VEL
LIN {X 0,Y 495.756,Z 288.725,A -85,B 0,C 180,E1 -6151.725,E2 -6151.725} C_VEL
LIN {X 0,Y 495.764,Z 288.729,A -85,B 0,C 180,E1 -6154.693,E2 -6154.693} C_VEL
LIN {X 0,Y 495.731,Z 288.732,A -85,B 0,C 180,E1 -6157.562,E2 -6157.562} C_VEL
LIN {X 0,Y 495.768,Z 288.727,A -85,B 0,C 180,E1 -6160.7,E2 -6160.7} C_VEL
LIN {X 0,Y 495.729,Z 288.732,A -85,B 0,C 180,E1 -6164.002,E2 -6164.002} C_VEL
LIN {X 0,Y 495.727,Z 288.735,A -85,B 0,C 180,E1 -6167.117,E2 -6167.117} C_VEL
LIN {X 0,Y 495.761,Z 288.73,A -85,B 0,C 180,E1 -6169.953,E2 -6169.953} C_VEL
LIN {X 0,Y 495.73,Z 288.732,A -85,B 0,C 180,E1 -6172.553,E2 -6172.553} C_VEL
LIN {X 0,Y 495.78,Z 288.732,A -85,B 0,C 180,E1 -6175.457,E2 -6175.457} C_VEL
LIN {X 0,Y 495.758,Z 288.731,A -85,B 0,C 180,E1 -6178.364,E2 -6178.364} C_VEL
LIN {X 0,Y 495.789,Z 288.728,A -85,B 0,C 180,E1 -6181.507,E2 -6181.507} C_VEL
LIN {X 0,Y 495.794,Z 288.732,A -85,B 0,C 180,E1 -6183.932,E2 -6183.932} C_VEL
LIN {X 0,Y 495.828,Z 288.749,A -85,B 0,C 180,E1 -6185.021,E2 -6185.021} C_VEL
LIN {X 0,Y 497.404,Z 298.59,A -85,B 0,C 180,E1 -6186.695,E2 -6186.695} C_VEL
LIN {X 0,Y 496.907,Z 317.531,A -85,B 0,C 180,E1 -6189.725,E2 -6189.725} C_VEL
LIN {X 0,Y 496.409,Z 336.311,A -85,B 0,C 180,E1 -6192.703,E2 -6192.703} C_VEL
LIN {X 0,Y 496.234,Z 344.424,A -85,B 0,C 180,E1 -6193.964,E2 -6193.964} C_VEL
LIN {X 0,Y 498.454,Z 359.221,A -85,B 0,C 180,E1 -6194.26,E2 -6194.26} C_VEL
LIN {X 0,Y 497.86,Z 453.151,A -85,B 0,C 180,E1 -6195.671,E2 -6195.671} C_VEL
LIN {X 0,Y 497.538,Z 466.301,A -85,B 0,C 180,E1 -6196.027,E2 -6196.027} C_VEL
LIN {X 0,Y 497.202,Z 479.555,A -85,B 0,C 180,E1 -6196.564,E2 -6196.564} C_VEL
LIN {X 0,Y 496.861,Z 491.495,A -85,B 0,C 180,E1 -6197.23,E2 -6197.23} C_VEL
LIN {X 0,Y 496.505,Z 502.991,A -85,B 0,C 180,E1 -6198.052,E2 -6198.052} C_VEL
LIN {X 0,Y 496.133,Z 513.352,A -85,B 0,C 180,E1 -6198.975,E2 -6198.975} C_VEL
LIN {X 0,Y 495.756,Z 522.656,A -85,B 0,C 180,E1 -6199.999,E2 -6199.999} C_VEL
LIN {X 0,Y 495.463,Z 531.705,A -85,B 0,C 180,E1 -6201.229,E2 -6201.229} C_VEL
LIN {X 0,Y 495.277,Z 538.995,A -85,B 0,C 180,E1 -6202.457,E2 -6202.457} C_VEL
LIN {X 0,Y 495.122,Z 545.12,A -85,B 0,C 180,E1 -6203.76,E2 -6203.76} C_VEL
LIN {X 0,Y 495.036,Z 550.024,A -85,B 0,C 180,E1 -6205.113,E2 -6205.113} C_VEL
LIN {X 0,Y 495.033,Z 552.35,A -85,B 0,C 180,E1 -6205.929,E2 -6205.929} C_VEL
LIN {X 0,Y 495.042,Z 554.238,A -85,B 0,C 180,E1 -6206.744,E2 -6206.744} C_VEL
LIN {X 0,Y 494.998,Z 555.652,A -85,B 0,C 180,E1 -6207.558,E2 -6207.558} C_VEL
LIN {X 0,Y 494.962,Z 556.663,A -85,B 0,C 180,E1 -6208.372,E2 -6208.372} C_VEL
LIN {X 0,Y 494.901,Z 557.506,A -85,B 0,C 180,E1 -6210,E2 -6210} C_VEL
LIN {X 0,Y 494.962,Z 556.688,A -85,B 0,C 180,E1 -6211.627,E2 -6211.627} C_VEL
LIN {X 0,Y 494.997,Z 555.691,A -85,B 0,C 180,E1 -6212.441,E2 -6212.441} C_VEL
LIN {X 0,Y 495.041,Z 554.288,A -85,B 0,C 180,E1 -6213.255,E2 -6213.255} C_VEL
LIN {X 0,Y 495.007,Z 551.332,A -85,B 0,C 180,E1 -6214.478,E2 -6214.478} C_VEL
LIN {X 0,Y 495.124,Z 547.333,A -85,B 0,C 180,E1 -6215.702,E2 -6215.702} C_VEL
LIN {X 0,Y 495.252,Z 541.171,A -85,B 0,C 180,E1 -6217.132,E2 -6217.132} C_VEL
LIN {X 0,Y 495.421,Z 534.441,A -85,B 0,C 180,E1 -6218.36,E2 -6218.36} C_VEL
LIN {X 0,Y 495.675,Z 526.09,A -85,B 0,C 180,E1 -6219.59,E2 -6219.59} C_VEL
LIN {X 0,Y 495.963,Z 517.504,A -85,B 0,C 180,E1 -6220.615,E2 -6220.615} C_VEL
LIN {X 0,Y 496.417,Z 506.912,A -85,B 0,C 180,E1 -6221.638,E2 -6221.638} C_VEL
LIN {X 0,Y 496.767,Z 495.421,A -85,B 0,C 180,E1 -6222.531,E2 -6222.531} C_VEL
LIN {X 0,Y 497.074,Z 484.864,A -85,B 0,C 180,E1 -6223.178,E2 -6223.178} C_VEL
LIN {X 0,Y 497.411,Z 472.89,A -85,B 0,C 180,E1 -6223.741,E2 -6223.741} C_VEL
LIN {X 0,Y 497.747,Z 459.975,A -85,B 0,C 180,E1 -6224.175,E2 -6224.175} C_VEL
LIN {X 0,Y 497.972,Z 446.338,A -85,B 0,C 180,E1 -6224.455,E2 -6224.455} C_VEL
LIN {X 0,Y 498.473,Z 359.234,A -85,B 0,C 180,E1 -6225.742,E2 -6225.742} C_VEL
LIN {X 0,Y 496.261,Z 344.819,A -85,B 0,C 180,E1 -6226.035,E2 -6226.035} C_VEL
LIN {X 0,Y 496.858,Z 325.338,A -85,B 0,C 180,E1 -6229.199,E2 -6229.199} C_VEL
LIN {X 0,Y 497.476,Z 307.112,A -85,B 0,C 180,E1 -6232.203,E2 -6232.203} C_VEL
LIN {X 0,Y 497.746,Z 299.949,A -85,B 0,C 180,E1 -6233.396,E2 -6233.396} C_VEL
LIN {X 0,Y 496.639,Z 292.966,A -85,B 0,C 180,E1 -6234.633,E2 -6234.633} C_VEL
LIN {X 0,Y 495.823,Z 288.726,A -85,B 0,C 180,E1 -6235.445,E2 -6235.445} C_VEL
LIN {X 0,Y 495.787,Z 288.726,A -85,B 0,C 180,E1 -6238.493,E2 -6238.493} C_VEL
LIN {X 0,Y 495.754,Z 288.729,A -85,B 0,C 180,E1 -6241.725,E2 -6241.725} C_VEL
LIN {X 0,Y 495.767,Z 288.727,A -85,B 0,C 180,E1 -6244.693,E2 -6244.693} C_VEL
LIN {X 0,Y 495.726,Z 288.73,A -85,B 0,C 180,E1 -6247.561,E2 -6247.561} C_VEL
LIN {X 0,Y 495.764,Z 288.729,A -85,B 0,C 180,E1 -6250.699,E2 -6250.699} C_VEL
LIN {X 0,Y 495.731,Z 288.732,A -85,B 0,C 180,E1 -6254,E2 -6254} C_VEL
LIN {X 0,Y 495.73,Z 288.731,A -85,B 0,C 180,E1 -6257.117,E2 -6257.117} C_VEL
LIN {X 0,Y 495.755,Z 288.727,A -85,B 0,C 180,E1 -6259.952,E2 -6259.952} C_VEL
LIN {X 0,Y 495.728,Z 288.736,A -85,B 0,C 180,E1 -6262.552,E2 -6262.552} C_VEL
LIN {X 0,Y 495.778,Z 288.724,A -85,B 0,C 180,E1 -6265.457,E2 -6265.457} C_VEL
LIN {X 0,Y 495.754,Z 288.728,A -85,B 0,C 180,E1 -6268.364,E2 -6268.364} C_VEL
LIN {X 0,Y 495.782,Z 288.724,A -85,B 0,C 180,E1 -6271.506,E2 -6271.506} C_VEL
LIN {X 0,Y 495.785,Z 288.722,A -85,B 0,C 180,E1 -6273.932,E2 -6273.932} C_VEL
LIN {X 0,Y 495.756,Z 288.735,A -85,B 0,C 180,E1 -6277.139,E2 -6277.139} C_VEL
LIN {X 0,Y 495.765,Z 288.725,A -85,B 0,C 180,E1 -6280.109,E2 -6280.109} C_VEL
LIN {X 0,Y 495.78,Z 288.724,A -85,B 0,C 180,E1 -6282.681,E2 -6282.681} C_VEL
LIN {X 0,Y 495.788,Z 288.73,A -85,B 0,C 180,E1 -6285.217,E2 -6285.217} C_VEL
LIN {X 0,Y 495.845,Z 288.715,A -85,B 0,C 180,E1 -6288.555,E2 -6288.555} C_VEL
LIN {X 0,Y 495.867,Z 288.716,A -85,B 0,C 180,E1 -6291.852,E2 -6291.852} C_VEL
LIN {X 0,Y 495.889,Z 288.71,A -85,B 0,C 180,E1 -6294.307,E2 -6294.307} C_VEL
LIN {X 0,Y 495.986,Z 288.705,A -85,B 0,C 180,E1 -6297.564,E2 -6297.564} C_VEL
LIN {X 0,Y 495.991,Z 288.702,A -85,B 0,C 180,E1 -6300,E2 -6300} C_VEL
LIN {X 0,Y 495.986,Z 288.698,A -85,B 0,C 180,E1 -6302.437,E2 -6302.437} C_VEL
LIN {X 0,Y 495.877,Z 288.717,A -85,B 0,C 180,E1 -6305.694,E2 -6305.694} C_VEL
LIN {X 0,Y 495.836,Z 288.716,A -85,B 0,C 180,E1 -6308.97,E2 -6308.97} C_VEL
LIN {X 0,Y 495.823,Z 288.727,A -85,B 0,C 180,E1 -6312.035,E2 -6312.035} C_VEL
LIN {X 0,Y 495.818,Z 288.719,A -85,B 0,C 180,E1 -6315.452,E2 -6315.452} C_VEL
LIN {X 0,Y 495.773,Z 288.733,A -85,B 0,C 180,E1 -6318.238,E2 -6318.238} C_VEL
LIN {X 0,Y 495.769,Z 288.727,A -85,B 0,C 180,E1 -6320.757,E2 -6320.757} C_VEL
LIN {X 0,Y 495.737,Z 288.728,A -85,B 0,C 180,E1 -6323.388,E2 -6323.388} C_VEL
LIN {X 0,Y 495.757,Z 288.73,A -85,B 0,C 180,E1 -6326.07,E2 -6326.07} C_VEL
LIN {X 0,Y 495.74,Z 288.732,A -85,B 0,C 180,E1 -6328.817,E2 -6328.817} C_VEL
LIN {X 0,Y 495.751,Z 288.726,A -85,B 0,C 180,E1 -6331.726,E2 -6331.726} C_VEL
LIN {X 0,Y 495.765,Z 288.734,A -85,B 0,C 180,E1 -6334.695,E2 -6334.695} C_VEL
LIN {X 0,Y 495.725,Z 288.73,A -85,B 0,C 180,E1 -6337.563,E2 -6337.563} C_VEL
LIN {X 0,Y 495.745,Z 288.735,A -85,B 0,C 180,E1 -6340.703,E2 -6340.703} C_VEL
LIN {X 0,Y 495.715,Z 288.731,A -85,B 0,C 180,E1 -6343.694,E2 -6343.694} C_VEL
LIN {X 0,Y 495.715,Z 288.732,A -85,B 0,C 180,E1 -6346.308,E2 -6346.308} C_VEL
LIN {X 0,Y 495.73,Z 288.735,A -85,B 0,C 180,E1 -6349.297,E2 -6349.297} C_VEL
LIN {X 0,Y 495.745,Z 288.732,A -85,B 0,C 180,E1 -6351.409,E2 -6351.409} C_VEL
LIN {X 0,Y 495.744,Z 288.728,A -85,B 0,C 180,E1 -6354.463,E2 -6354.463} C_VEL
LIN {X 0,Y 495.765,Z 288.732,A -85,B 0,C 180,E1 -6357.406,E2 -6357.406} C_VEL
LIN {X 0,Y 495.757,Z 288.726,A -85,B 0,C 180,E1 -6360.254,E2 -6360.254} C_VEL
LIN {X 0,Y 495.726,Z 288.731,A -85,B 0,C 180,E1 -6360.739,E2 -6360.739} C_VEL
LIN {X 0,Y 495.047,Z 288.823,A -85,B 0,C 180,E1 -6361.418,E2 -6361.418} C_VEL
LIN {X 0,Y 492.171,Z 289.178,A -85,B 0,C 180,E1 -6362.52,E2 -6362.52} C_VEL
LIN {X 0,Y 489.754,Z 289.482,A -85,B 0,C 180,E1 -6363.408,E2 -6363.408} C_VEL
LIN {X 0,Y 488.731,Z 289.603,A -85,B 0,C 180,E1 -6364.094,E2 -6364.094} C_VEL
LIN {X 0,Y 488.655,Z 289.61,A -85,B 0,C 180,E1 -6364.326,E2 -6364.326} C_VEL
LIN {X 0,Y 488.724,Z 289.605,A -85,B 0,C 180,E1 -6367.154,E2 -6367.154} C_VEL
LIN {X 0,Y 488.719,Z 289.609,A -85,B 0,C 180,E1 -6369.811,E2 -6369.811} C_VEL
LIN {X 0,Y 488.694,Z 289.606,A -85,B 0,C 180,E1 -6372.423,E2 -6372.423} C_VEL
LIN {X 0,Y 488.764,Z 289.597,A -85,B 0,C 180,E1 -6375,E2 -6375} C_VEL
LIN {X 0,Y 488.787,Z 289.596,A -85,B 0,C 180,E1 -6378.388,E2 -6378.388} C_VEL
LIN {X 0,Y 488.758,Z 289.603,A -85,B 0,C 180,E1 -6381.733,E2 -6381.733} C_VEL
LIN {X 0,Y 488.815,Z 289.597,A -85,B 0,C 180,E1 -6384.224,E2 -6384.224} C_VEL
LIN {X 0,Y 488.937,Z 289.577,A -85,B 0,C 180,E1 -6387.529,E2 -6387.529} C_VEL
LIN {X 0,Y 488.944,Z 289.581,A -85,B 0,C 180,E1 -6390,E2 -6390} C_VEL
LIN {X 0,Y 488.936,Z 289.581,A -85,B 0,C 180,E1 -6392.472,E2 -6392.472} C_VEL
LIN {X 0,Y 488.813,Z 289.592,A -85,B 0,C 180,E1 -6395.777,E2 -6395.777} C_VEL
LIN {X 0,Y 488.758,Z 289.605,A -85,B 0,C 180,E1 -6398.268,E2 -6398.268} C_VEL
LIN {X 0,Y 488.761,Z 289.597,A -85,B 0,C 180,E1 -6401.614,E2 -6401.614} C_VEL
LIN {X 0,Y 488.718,Z 289.606,A -85,B 0,C 180,E1 -6405.002,E2 -6405.002} C_VEL
LIN {X 0,Y 488.711,Z 289.609,A -85,B 0,C 180,E1 -6408.444,E2 -6408.444} C_VEL
LIN {X 0,Y 488.704,Z 289.611,A -85,B 0,C 180,E1 -6411.071,E2 -6411.071} C_VEL
LIN {X 0,Y 488.663,Z 289.613,A -85,B 0,C 180,E1 -6413.747,E2 -6413.747} C_VEL
LIN {X 0,Y 488.733,Z 289.769,A -85,B 0,C 180,E1 -6416.574,E2 -6416.574} C_VEL
LIN {X 0,Y 489.648,Z 295.554,A -85,B 0,C 180,E1 -6417.806,E2 -6417.806} C_VEL
LIN {X 0,Y 489.299,Z 310.316,A -85,B 0,C 180,E1 -6420.791,E2 -6420.791} C_VEL
LIN {X 0,Y 491.74,Z 323.15,A -85,B 0,C 180,E1 -6421.085,E2 -6421.085} C_VEL
LIN {X 0,Y 491.076,Z 417.721,A -85,B 0,C 180,E1 -6422.529,E2 -6422.529} C_VEL
LIN {X 0,Y 490.806,Z 431.006,A -85,B 0,C 180,E1 -6422.901,E2 -6422.901} C_VEL
LIN {X 0,Y 490.511,Z 443.466,A -85,B 0,C 180,E1 -6423.417,E2 -6423.417} C_VEL
LIN {X 0,Y 490.084,Z 456.019,A -85,B 0,C 180,E1 -6424.13,E2 -6424.13} C_VEL
LIN {X 0,Y 489.737,Z 466.655,A -85,B 0,C 180,E1 -6424.906,E2 -6424.906} C_VEL
LIN {X 0,Y 489.381,Z 476.751,A -85,B 0,C 180,E1 -6425.818,E2 -6425.818} C_VEL
LIN {X 0,Y 488.963,Z 486.78,A -85,B 0,C 180,E1 -6426.944,E2 -6426.944} C_VEL
LIN {X 0,Y 488.622,Z 495.784,A -85,B 0,C 180,E1 -6428.206,E2 -6428.206} C_VEL
LIN {X 0,Y 488.342,Z 503.313,A -85,B 0,C 180,E1 -6429.531,E2 -6429.531} C_VEL
LIN {X 0,Y 488.178,Z 509.48,A -85,B 0,C 180,E1 -6430.923,E2 -6430.923} C_VEL
LIN {X 0,Y 488.05,Z 513.362,A -85,B 0,C 180,E1 -6432.037,E2 -6432.037} C_VEL
LIN {X 0,Y 487.964,Z 516.518,A -85,B 0,C 180,E1 -6433.206,E2 -6433.206} C_VEL
LIN {X 0,Y 487.928,Z 518.011,A -85,B 0,C 180,E1 -6433.929,E2 -6433.929} C_VEL
LIN {X 0,Y 487.867,Z 519.778,A -85,B 0,C 180,E1 -6435.099,E2 -6435.099} C_VEL
LIN {X 0,Y 487.809,Z 520.694,A -85,B 0,C 180,E1 -6436.247,E2 -6436.247} C_VEL
LIN {X 0,Y 487.835,Z 520.844,A -85,B 0,C 180,E1 -6437.382,E2 -6437.382} C_VEL
LIN {X 0,Y 487.849,Z 520.268,A -85,B 0,C 180,E1 -6438.514,E2 -6438.514} C_VEL
LIN {X 0,Y 487.875,Z 518.74,A -85,B 0,C 180,E1 -6439.772,E2 -6439.772} C_VEL
LIN {X 0,Y 487.949,Z 516.183,A -85,B 0,C 180,E1 -6441.057,E2 -6441.057} C_VEL
LIN {X 0,Y 488.076,Z 512.455,A -85,B 0,C 180,E1 -6442.37,E2 -6442.37} C_VEL
LIN {X 0,Y 488.267,Z 506.847,A -85,B 0,C 180,E1 -6443.832,E2 -6443.832} C_VEL
LIN {X 0,Y 488.469,Z 500.618,A -85,B 0,C 180,E1 -6445.096,E2 -6445.096} C_VEL
LIN {X 0,Y 488.704,Z 493.757,A -85,B 0,C 180,E1 -6446.222,E2 -6446.222} C_VEL
LIN {X 0,Y 489.06,Z 484.981,A -85,B 0,C 180,E1 -6447.391,E2 -6447.391} C_VEL
LIN {X 0,Y 489.43,Z 474.539,A -85,B 0,C 180,E1 -6448.511,E2 -6448.511} C_VEL
LIN {X 0,Y 489.861,Z 464.107,A -85,B 0,C 180,E1 -6449.408,E2 -6449.408} C_VEL
LIN {X 0,Y 490.268,Z 452.74,A -85,B 0,C 180,E1 -6450.182,E2 -6450.182} C_VEL
LIN {X 0,Y 490.646,Z 441.079,A -85,B 0,C 180,E1 -6450.796,E2 -6450.796} C_VEL
LIN {X 0,Y 490.83,Z 428.415,A -85,B 0,C 180,E1 -6451.292,E2 -6451.292} C_VEL
LIN {X 0,Y 491.09,Z 415.466,A -85,B 0,C 180,E1 -6451.615,E2 -6451.615} C_VEL
LIN {X 0,Y 491.689,Z 322.545,A -85,B 0,C 180,E1 -6453.031,E2 -6453.031} C_VEL
LIN {X 0,Y 489.292,Z 309.711,A -85,B 0,C 180,E1 -6453.331,E2 -6453.331} C_VEL
LIN {X 0,Y 489.382,Z 293.621,A -85,B 0,C 180,E1 -6456.065,E2 -6456.065} C_VEL
LIN {X 0,Y 488.767,Z 289.605,A -85,B 0,C 180,E1 -6456.787,E2 -6456.787} C_VEL
LIN {X 0,Y 488.727,Z 289.607,A -85,B 0,C 180,E1 -6459.81,E2 -6459.81} C_VEL
LIN {X 0,Y 488.717,Z 289.608,A -85,B 0,C 180,E1 -6462.422,E2 -6462.422} C_VEL
LIN {X 0,Y 488.767,Z 289.604,A -85,B 0,C 180,E1 -6464.999,E2 -6464.999} C_VEL
LIN {X 0,Y 488.807,Z 289.593,A -85,B 0,C 180,E1 -6468.387,E2 -6468.387} C_VEL
LIN {X 0,Y 488.817,Z 289.598,A -85,B 0,C 180,E1 -6471.733,E2 -6471.733} C_VEL
LIN {X 0,Y 488.848,Z 289.591,A -85,B 0,C 180,E1 -6474.224,E2 -6474.224} C_VEL
LIN {X 0,Y 488.961,Z 289.578,A -85,B 0,C 180,E1 -6477.528,E2 -6477.528} C_VEL
LIN {X 0,Y 488.935,Z 289.575,A -85,B 0,C 180,E1 -6480.823,E2 -6480.823} C_VEL
LIN {X 0,Y 488.962,Z 289.576,A -85,B 0,C 180,E1 -6482.471,E2 -6482.471} C_VEL
LIN {X 0,Y 488.839,Z 289.593,A -85,B 0,C 180,E1 -6485.776,E2 -6485.776} C_VEL
LIN {X 0,Y 488.818,Z 289.599,A -85,B 0,C 180,E1 -6488.266,E2 -6488.266} C_VEL
LIN {X 0,Y 488.807,Z 289.593,A -85,B 0,C 180,E1 -6491.612,E2 -6491.612} C_VEL
LIN {X 0,Y 488.766,Z 289.599,A -85,B 0,C 180,E1 -6495,E2 -6495} C_VEL
LIN {X 0,Y 488.748,Z 289.605,A -85,B 0,C 180,E1 -6498.442,E2 -6498.442} C_VEL
LIN {X 0,Y 488.708,Z 289.606,A -85,B 0,C 180,E1 -6501.071,E2 -6501.071} C_VEL
LIN {X 0,Y 488.69,Z 289.605,A -85,B 0,C 180,E1 -6503.746,E2 -6503.746} C_VEL
LIN {X 0,Y 488.793,Z 289.598,A -85,B 0,C 180,E1 -6506.943,E2 -6506.943} C_VEL
LIN {X 0,Y 488.711,Z 289.606,A -85,B 0,C 180,E1 -6510.363,E2 -6510.363} C_VEL
LIN {X 0,Y 488.73,Z 289.604,A -85,B 0,C 180,E1 -6513.483,E2 -6513.483} C_VEL
LIN {X 0,Y 488.684,Z 289.609,A -85,B 0,C 180,E1 -6516.354,E2 -6516.354} C_VEL
LIN {X 0,Y 488.703,Z 289.614,A -85,B 0,C 180,E1 -6519.254,E2 -6519.254} C_VEL
LIN {X 0,Y 488.709,Z 289.61,A -85,B 0,C 180,E1 -6521.6,E2 -6521.6} C_VEL
LIN {X 0,Y 488.703,Z 289.608,A -85,B 0,C 180,E1 -6524.803,E2 -6524.803} C_VEL
LIN {X 0,Y 488.694,Z 289.614,A -85,B 0,C 180,E1 -6527.474,E2 -6527.474} C_VEL
LIN {X 0,Y 488.735,Z 289.608,A -85,B 0,C 180,E1 -6529.677,E2 -6529.677} C_VEL
LIN {X 0,Y 488.681,Z 289.611,A -85,B 0,C 180,E1 -6532.841,E2 -6532.841} C_VEL
LIN {X 0,Y 488.733,Z 289.612,A -85,B 0,C 180,E1 -6535.887,E2 -6535.887} C_VEL
LIN {X 0,Y 488.695,Z 289.609,A -85,B 0,C 180,E1 -6538.82,E2 -6538.82} C_VEL
LIN {X 0,Y 488.746,Z 289.607,A -85,B 0,C 180,E1 -6541.671,E2 -6541.671} C_VEL
LIN {X 0,Y 488.757,Z 289.607,A -85,B 0,C 180,E1 -6544.445,E2 -6544.445} C_VEL
LIN {X 0,Y 488.781,Z 289.64,A -85,B 0,C 180,E1 -6544.847,E2 -6544.847} C_VEL
LIN {X 0,Y 490.444,Z 299.248,A -85,B 0,C 180,E1 -6546.508,E2 -6546.508} C_VEL
LIN {X 0,Y 489.981,Z 317.213,A -85,B 0,C 180,E1 -6549.426,E2 -6549.426} C_VEL
LIN {X 0,Y 489.416,Z 336.009,A -85,B 0,C 180,E1 -6552.448,E2 -6552.448} C_VEL
LIN {X 0,Y 489.232,Z 344.193,A -85,B 0,C 180,E1 -6553.727,E2 -6553.727} C_VEL
LIN {X 0,Y 491.627,Z 360.715,A -85,B 0,C 180,E1 -6554.064,E2 -6554.064} C_VEL
LIN {X 0,Y 490.974,Z 452.701,A -85,B 0,C 180,E1 -6555.466,E2 -6555.466} C_VEL
LIN {X 0,Y 490.634,Z 465.898,A -85,B 0,C 180,E1 -6555.826,E2 -6555.826} C_VEL
LIN {X 0,Y 490.287,Z 479.185,A -85,B 0,C 180,E1 -6556.371,E2 -6556.371} C_VEL
LIN {X 0,Y 489.908,Z 491.129,A -85,B 0,C 180,E1 -6557.045,E2 -6557.045} C_VEL
LIN {X 0,Y 489.496,Z 502.657,A -85,B 0,C 180,E1 -6557.878,E2 -6557.878} C_VEL
LIN {X 0,Y 489.095,Z 513.032,A -85,B 0,C 180,E1 -6558.814,E2 -6558.814} C_VEL
LIN {X 0,Y 488.727,Z 522.346,A -85,B 0,C 180,E1 -6559.854,E2 -6559.854} C_VEL
LIN {X 0,Y 488.406,Z 531.401,A -85,B 0,C 180,E1 -6561.101,E2 -6561.101} C_VEL
LIN {X 0,Y 488.209,Z 538.699,A -85,B 0,C 180,E1 -6562.347,E2 -6562.347} C_VEL
LIN {X 0,Y 488.049,Z 544.231,A -85,B 0,C 180,E1 -6563.522,E2 -6563.522} C_VEL
LIN {X 0,Y 488.018,Z 548.413,A -85,B 0,C 180,E1 -6564.628,E2 -6564.628} C_VEL
LIN {X 0,Y 487.929,Z 552.073,A -85,B 0,C 180,E1 -6565.87,E2 -6565.87} C_VEL
LIN {X 0,Y 487.964,Z 553.966,A -85,B 0,C 180,E1 -6566.697,E2 -6566.697} C_VEL
LIN {X 0,Y 487.908,Z 555.384,A -85,B 0,C 180,E1 -6567.523,E2 -6567.523} C_VEL
LIN {X 0,Y 487.89,Z 556.397,A -85,B 0,C 180,E1 -6568.349,E2 -6568.349} C_VEL
LIN {X 0,Y 487.821,Z 557.243,A -85,B 0,C 180,E1 -6570,E2 -6570} C_VEL
LIN {X 0,Y 487.89,Z 556.426,A -85,B 0,C 180,E1 -6571.65,E2 -6571.65} C_VEL
LIN {X 0,Y 487.908,Z 555.427,A -85,B 0,C 180,E1 -6572.476,E2 -6572.476} C_VEL
LIN {X 0,Y 487.964,Z 554.023,A -85,B 0,C 180,E1 -6573.302,E2 -6573.302} C_VEL
LIN {X 0,Y 487.92,Z 551.065,A -85,B 0,C 180,E1 -6574.543,E2 -6574.543} C_VEL
LIN {X 0,Y 488.021,Z 547.061,A -85,B 0,C 180,E1 -6575.785,E2 -6575.785} C_VEL
LIN {X 0,Y 488.179,Z 540.892,A -85,B 0,C 180,E1 -6577.236,E2 -6577.236} C_VEL
LIN {X 0,Y 488.352,Z 534.154,A -85,B 0,C 180,E1 -6578.482,E2 -6578.482} C_VEL
LIN {X 0,Y 488.617,Z 525.791,A -85,B 0,C 180,E1 -6579.729,E2 -6579.729} C_VEL
LIN {X 0,Y 488.957,Z 517.189,A -85,B 0,C 180,E1 -6580.769,E2 -6580.769} C_VEL
LIN {X 0,Y 489.432,Z 506.576,A -85,B 0,C 180,E1 -6581.807,E2 -6581.807} C_VEL
LIN {X 0,Y 489.762,Z 496.15,A -85,B 0,C 180,E1 -6582.633,E2 -6582.633} C_VEL
LIN {X 0,Y 490.12,Z 484.458,A -85,B 0,C 180,E1 -6583.368,E2 -6583.368} C_VEL
LIN {X 0,Y 490.515,Z 472.43,A -85,B 0,C 180,E1 -6583.938,E2 -6583.938} C_VEL
LIN {X 0,Y 490.843,Z 459.428,A -85,B 0,C 180,E1 -6584.378,E2 -6584.378} C_VEL
LIN {X 0,Y 491.085,Z 445.53,A -85,B 0,C 180,E1 -6584.662,E2 -6584.662} C_VEL
LIN {X 0,Y 491.573,Z 359.598,A -85,B 0,C 180,E1 -6585.956,E2 -6585.956} C_VEL
LIN {X 0,Y 489.293,Z 344.602,A -85,B 0,C 180,E1 -6586.264,E2 -6586.264} C_VEL
LIN {X 0,Y 489.917,Z 325.096,A -85,B 0,C 180,E1 -6589.482,E2 -6589.482} C_VEL
LIN {X 0,Y 490.631,Z 306.867,A -85,B 0,C 180,E1 -6592.53,E2 -6592.53} C_VEL
LIN {X 0,Y 490.754,Z 300.351,A -85,B 0,C 180,E1 -6593.639,E2 -6593.639} C_VEL
LIN {X 0,Y 488.788,Z 289.602,A -85,B 0,C 180,E1 -6595.61,E2 -6595.61} C_VEL
LIN {X 0,Y 488.744,Z 289.606,A -85,B 0,C 180,E1 -6598.328,E2 -6598.328} C_VEL
LIN {X 0,Y 488.69,Z 289.606,A -85,B 0,C 180,E1 -6601.179,E2 -6601.179} C_VEL
LIN {X 0,Y 488.728,Z 289.609,A -85,B 0,C 180,E1 -6604.112,E2 -6604.112} C_VEL
LIN {X 0,Y 488.677,Z 289.608,A -85,B 0,C 180,E1 -6607.158,E2 -6607.158} C_VEL
LIN {X 0,Y 488.715,Z 289.612,A -85,B 0,C 180,E1 -6610.344,E2 -6610.344} C_VEL
LIN {X 0,Y 488.684,Z 289.607,A -85,B 0,C 180,E1 -6613.654,E2 -6613.654} C_VEL
LIN {X 0,Y 488.689,Z 289.613,A -85,B 0,C 180,E1 -6616.346,E2 -6616.346} C_VEL
LIN {X 0,Y 488.716,Z 289.612,A -85,B 0,C 180,E1 -6618.585,E2 -6618.585} C_VEL
LIN {X 0,Y 488.677,Z 289.608,A -85,B 0,C 180,E1 -6621.8,E2 -6621.8} C_VEL
LIN {X 0,Y 488.723,Z 289.607,A -85,B 0,C 180,E1 -6625.051,E2 -6625.051} C_VEL
LIN {X 0,Y 488.701,Z 289.605,A -85,B 0,C 180,E1 -6628.045,E2 -6628.045} C_VEL
LIN {X 0,Y 488.718,Z 289.609,A -85,B 0,C 180,E1 -6630.729,E2 -6630.729} C_VEL
LIN {X 0,Y 488.751,Z 289.6,A -85,B 0,C 180,E1 -6633.528,E2 -6633.528} C_VEL
LIN {X 0,Y 488.687,Z 289.607,A -85,B 0,C 180,E1 -6636.254,E2 -6636.254} C_VEL
LIN {X 0,Y 488.74,Z 289.609,A -85,B 0,C 180,E1 -6639.175,E2 -6639.175} C_VEL
LIN {X 0,Y 488.728,Z 289.602,A -85,B 0,C 180,E1 -6642.423,E2 -6642.423} C_VEL
LIN {X 0,Y 488.759,Z 289.602,A -85,B 0,C 180,E1 -6645,E2 -6645} C_VEL
LIN {X 0,Y 488.799,Z 289.592,A -85,B 0,C 180,E1 -6648.388,E2 -6648.388} C_VEL
LIN {X 0,Y 488.812,Z 289.596,A -85,B 0,C 180,E1 -6651.734,E2 -6651.734} C_VEL
LIN {X 0,Y 488.849,Z 289.587,A -85,B 0,C 180,E1 -6654.224,E2 -6654.224} C_VEL
LIN {X 0,Y 488.954,Z 289.581,A -85,B 0,C 180,E1 -6657.529,E2 -6657.529} C_VEL
LIN {X 0,Y 488.962,Z 289.577,A -85,B 0,C 180,E1 -6660,E2 -6660} C_VEL
LIN {X 0,Y 488.954,Z 289.574,A -85,B 0,C 180,E1 -6662.472,E2 -6662.472} C_VEL
LIN {X 0,Y 488.834,Z 289.596,A -85,B 0,C 180,E1 -6665.776,E2 -6665.776} C_VEL
LIN {X 0,Y 488.811,Z 289.595,A -85,B 0,C 180,E1 -6668.267,E2 -6668.267} C_VEL
LIN {X 0,Y 488.8,Z 289.595,A -85,B 0,C 180,E1 -6671.613,E2 -6671.613} C_VEL
LIN {X 0,Y 488.755,Z 289.598,A -85,B 0,C 180,E1 -6675.001,E2 -6675.001} C_VEL
LIN {X 0,Y 488.741,Z 289.605,A -85,B 0,C 180,E1 -6678.443,E2 -6678.443} C_VEL
LIN {X 0,Y 488.702,Z 289.605,A -85,B 0,C 180,E1 -6681.071,E2 -6681.071} C_VEL
LIN {X 0,Y 488.671,Z 289.61,A -85,B 0,C 180,E1 -6683.747,E2 -6683.747} C_VEL
LIN {X 0,Y 488.714,Z 289.612,A -85,B 0,C 180,E1 -6686.475,E2 -6686.475} C_VEL
LIN {X 0,Y 488.706,Z 289.605,A -85,B 0,C 180,E1 -6689.272,E2 -6689.272} C_VEL
LIN {X 0,Y 488.699,Z 289.608,A -85,B 0,C 180,E1 -6692.148,E2 -6692.148} C_VEL
LIN {X 0,Y 488.714,Z 289.606,A -85,B 0,C 180,E1 -6695.116,E2 -6695.116} C_VEL
LIN {X 0,Y 488.674,Z 289.61,A -85,B 0,C 180,E1 -6698.201,E2 -6698.201} C_VEL
LIN {X 0,Y 488.716,Z 289.605,A -85,B 0,C 180,E1 -6700.345,E2 -6700.345} C_VEL
LIN {X 0,Y 488.674,Z 289.609,A -85,B 0,C 180,E1 -6703.656,E2 -6703.656} C_VEL
LIN {X 0,Y 488.674,Z 289.609,A -85,B 0,C 180,E1 -6706.345,E2 -6706.345} C_VEL
LIN {X 0,Y 488.702,Z 289.606,A -85,B 0,C 180,E1 -6709.674,E2 -6709.674} C_VEL
LIN {X 0,Y 488.677,Z 289.612,A -85,B 0,C 180,E1 -6712.842,E2 -6712.842} C_VEL
LIN {X 0,Y 488.723,Z 289.603,A -85,B 0,C 180,E1 -6715.887,E2 -6715.887} C_VEL
LIN {X 0,Y 488.685,Z 289.609,A -85,B 0,C 180,E1 -6718.821,E2 -6718.821} C_VEL
LIN {X 0,Y 488.695,Z 289.611,A -85,B 0,C 180,E1 -6721.669,E2 -6721.669} C_VEL
LIN {X 0,Y 488.655,Z 289.61,A -85,B 0,C 180,E1 -6724.326,E2 -6724.326} C_VEL
LIN {X 0,Y 488.012,Z 289.694,A -85,B 0,C 180,E1 -6725.014,E2 -6725.014} C_VEL
LIN {X 0,Y 485.18,Z 290.05,A -85,B 0,C 180,E1 -6726.132,E2 -6726.132} C_VEL
LIN {X 0,Y 482.768,Z 290.353,A -85,B 0,C 180,E1 -6727.033,E2 -6727.033} C_VEL
LIN {X 0,Y 481.726,Z 290.48,A -85,B 0,C 180,E1 -6727.729,E2 -6727.729} C_VEL
LIN {X 0,Y 481.638,Z 290.488,A -85,B 0,C 180,E1 -6727.964,E2 -6727.964} C_VEL
LIN {X 0,Y 481.696,Z 290.478,A -85,B 0,C 180,E1 -6730.393,E2 -6730.393} C_VEL
LIN {X 0,Y 481.665,Z 290.482,A -85,B 0,C 180,E1 -6733.034,E2 -6733.034} C_VEL
LIN {X 0,Y 481.688,Z 290.485,A -85,B 0,C 180,E1 -6735.639,E2 -6735.639} C_VEL
LIN {X 0,Y 481.738,Z 290.476,A -85,B 0,C 180,E1 -6738.215,E2 -6738.215} C_VEL
LIN {X 0,Y 481.716,Z 290.479,A -85,B 0,C 180,E1 -6741.611,E2 -6741.611} C_VEL
LIN {X 0,Y 481.776,Z 290.475,A -85,B 0,C 180,E1 -6744.14,E2 -6744.14} C_VEL
LIN {X 0,Y 481.902,Z 290.453,A -85,B 0,C 180,E1 -6747.493,E2 -6747.493} C_VEL
LIN {X 0,Y 481.914,Z 290.457,A -85,B 0,C 180,E1 -6750,E2 -6750} C_VEL
LIN {X 0,Y 481.901,Z 290.457,A -85,B 0,C 180,E1 -6752.508,E2 -6752.508} C_VEL
LIN {X 0,Y 481.775,Z 290.47,A -85,B 0,C 180,E1 -6755.861,E2 -6755.861} C_VEL
LIN {X 0,Y 481.715,Z 290.484,A -85,B 0,C 180,E1 -6758.39,E2 -6758.39} C_VEL
LIN {X 0,Y 481.717,Z 290.475,A -85,B 0,C 180,E1 -6761.786,E2 -6761.786} C_VEL
LIN {X 0,Y 481.695,Z 290.479,A -85,B 0,C 180,E1 -6765.226,E2 -6765.226} C_VEL
LIN {X 0,Y 481.655,Z 290.491,A -85,B 0,C 180,E1 -6768.724,E2 -6768.724} C_VEL
LIN {X 0,Y 481.64,Z 290.488,A -85,B 0,C 180,E1 -6771.395,E2 -6771.395} C_VEL
LIN {X 0,Y 481.623,Z 290.491,A -85,B 0,C 180,E1 -6774.116,E2 -6774.116} C_VEL
LIN {X 0,Y 481.692,Z 290.675,A -85,B 0,C 180,E1 -6776.424,E2 -6776.424} C_VEL
LIN {X 0,Y 482.681,Z 296.909,A -85,B 0,C 180,E1 -6777.771,E2 -6777.771} C_VEL
LIN {X 0,Y 482.337,Z 310.571,A -85,B 0,C 180,E1 -6780.563,E2 -6780.563} C_VEL
LIN {X 0,Y 484.948,Z 324.517,A -85,B 0,C 180,E1 -6780.878,E2 -6780.878} C_VEL
LIN {X 0,Y 484.202,Z 418.027,A -85,B 0,C 180,E1 -6782.329,E2 -6782.329} C_VEL
LIN {X 0,Y 483.909,Z 431.264,A -85,B 0,C 180,E1 -6782.704,E2 -6782.704} C_VEL
LIN {X 0,Y 483.609,Z 443.593,A -85,B 0,C 180,E1 -6783.222,E2 -6783.222} C_VEL
LIN {X 0,Y 483.189,Z 455.522,A -85,B 0,C 180,E1 -6783.901,E2 -6783.901} C_VEL
LIN {X 0,Y 482.774,Z 466.689,A -85,B 0,C 180,E1 -6784.72,E2 -6784.72} C_VEL
LIN {X 0,Y 482.417,Z 476.808,A -85,B 0,C 180,E1 -6785.643,E2 -6785.643} C_VEL
LIN {X 0,Y 482.011,Z 486.327,A -85,B 0,C 180,E1 -6786.713,E2 -6786.713} C_VEL
LIN {X 0,Y 481.597,Z 495.487,A -85,B 0,C 180,E1 -6787.998,E2 -6787.998} C_VEL
LIN {X 0,Y 481.318,Z 502.914,A -85,B 0,C 180,E1 -6789.295,E2 -6789.295} C_VEL
LIN {X 0,Y 481.142,Z 508.72,A -85,B 0,C 180,E1 -6790.574,E2 -6790.574} C_VEL
LIN {X 0,Y 480.982,Z 513.19,A -85,B 0,C 180,E1 -6791.823,E2 -6791.823} C_VEL
LIN {X 0,Y 480.874,Z 517.271,A -85,B 0,C 180,E1 -6793.386,E2 -6793.386} C_VEL
LIN {X 0,Y 480.799,Z 519.361,A -85,B 0,C 180,E1 -6794.558,E2 -6794.558} C_VEL
LIN {X 0,Y 480.758,Z 520.673,A -85,B 0,C 180,E1 -6795.751,E2 -6795.751} C_VEL
LIN {X 0,Y 480.725,Z 521.156,A -85,B 0,C 180,E1 -6796.969,E2 -6796.969} C_VEL
LIN {X 0,Y 480.748,Z 520.775,A -85,B 0,C 180,E1 -6798.208,E2 -6798.208} C_VEL
LIN {X 0,Y 480.763,Z 519.487,A -85,B 0,C 180,E1 -6799.478,E2 -6799.478} C_VEL
LIN {X 0,Y 480.874,Z 516.581,A -85,B 0,C 180,E1 -6801.064,E2 -6801.064} C_VEL
LIN {X 0,Y 481.038,Z 511.956,A -85,B 0,C 180,E1 -6802.676,E2 -6802.676} C_VEL
LIN {X 0,Y 481.205,Z 507.428,A -85,B 0,C 180,E1 -6803.858,E2 -6803.858} C_VEL
LIN {X 0,Y 481.445,Z 500.438,A -85,B 0,C 180,E1 -6805.297,E2 -6805.297} C_VEL
LIN {X 0,Y 481.818,Z 492.409,A -85,B 0,C 180,E1 -6806.589,E2 -6806.589} C_VEL
LIN {X 0,Y 482.159,Z 483.758,A -85,B 0,C 180,E1 -6807.717,E2 -6807.717} C_VEL
LIN {X 0,Y 482.503,Z 474.429,A -85,B 0,C 180,E1 -6808.712,E2 -6808.712} C_VEL
LIN {X 0,Y 482.928,Z 463.913,A -85,B 0,C 180,E1 -6809.621,E2 -6809.621} C_VEL
LIN {X 0,Y 483.366,Z 452.944,A -85,B 0,C 180,E1 -6810.373,E2 -6810.373} C_VEL
LIN {X 0,Y 483.755,Z 441.279,A -85,B 0,C 180,E1 -6810.995,E2 -6810.995} C_VEL
LIN {X 0,Y 483.964,Z 428.557,A -85,B 0,C 180,E1 -6811.499,E2 -6811.499} C_VEL
LIN {X 0,Y 484.231,Z 415.52,A -85,B 0,C 180,E1 -6811.826,E2 -6811.826} C_VEL
LIN {X 0,Y 484.92,Z 323.7,A -85,B 0,C 180,E1 -6813.252,E2 -6813.252} C_VEL
LIN {X 0,Y 482.324,Z 309.927,A -85,B 0,C 180,E1 -6813.584,E2 -6813.584} C_VEL
LIN {X 0,Y 482.444,Z 294.844,A -85,B 0,C 180,E1 -6816.156,E2 -6816.156} C_VEL
LIN {X 0,Y 481.731,Z 290.482,A -85,B 0,C 180,E1 -6816.96,E2 -6816.96} C_VEL
LIN {X 0,Y 481.707,Z 290.48,A -85,B 0,C 180,E1 -6820.393,E2 -6820.393} C_VEL
LIN {X 0,Y 481.682,Z 290.489,A -85,B 0,C 180,E1 -6823.033,E2 -6823.033} C_VEL
LIN {X 0,Y 481.696,Z 290.488,A -85,B 0,C 180,E1 -6825.639,E2 -6825.639} C_VEL
LIN {X 0,Y 481.753,Z 290.473,A -85,B 0,C 180,E1 -6828.215,E2 -6828.215} C_VEL
LIN {X 0,Y 481.762,Z 290.477,A -85,B 0,C 180,E1 -6831.611,E2 -6831.611} C_VEL
LIN {X 0,Y 481.809,Z 290.469,A -85,B 0,C 180,E1 -6834.139,E2 -6834.139} C_VEL
LIN {X 0,Y 481.928,Z 290.454,A -85,B 0,C 180,E1 -6837.492,E2 -6837.492} C_VEL
LIN {X 0,Y 481.887,Z 290.452,A -85,B 0,C 180,E1 -6840.835,E2 -6840.835} C_VEL
LIN {X 0,Y 481.929,Z 290.452,A -85,B 0,C 180,E1 -6842.507,E2 -6842.507} C_VEL
LIN {X 0,Y 481.798,Z 290.471,A -85,B 0,C 180,E1 -6845.86,E2 -6845.86} C_VEL
LIN {X 0,Y 481.763,Z 290.476,A -85,B 0,C 180,E1 -6848.388,E2 -6848.388} C_VEL
LIN {X 0,Y 481.752,Z 290.473,A -85,B 0,C 180,E1 -6851.785,E2 -6851.785} C_VEL
LIN {X 0,Y 481.746,Z 290.473,A -85,B 0,C 180,E1 -6855.224,E2 -6855.224} C_VEL
LIN {X 0,Y 481.71,Z 290.483,A -85,B 0,C 180,E1 -6858.722,E2 -6858.722} C_VEL
LIN {X 0,Y 481.647,Z 290.483,A -85,B 0,C 180,E1 -6861.395,E2 -6861.395} C_VEL
LIN {X 0,Y 481.675,Z 290.481,A -85,B 0,C 180,E1 -6864.113,E2 -6864.113} C_VEL
LIN {X 0,Y 481.748,Z 290.473,A -85,B 0,C 180,E1 -6867.139,E2 -6867.139} C_VEL
LIN {X 0,Y 481.68,Z 290.48,A -85,B 0,C 180,E1 -6869.741,E2 -6869.741} C_VEL
LIN {X 0,Y 481.672,Z 290.484,A -85,B 0,C 180,E1 -6872.674,E2 -6872.674} C_VEL
LIN {X 0,Y 481.637,Z 290.487,A -85,B 0,C 180,E1 -6875.71,E2 -6875.71} C_VEL
LIN {X 0,Y 481.672,Z 290.484,A -85,B 0,C 180,E1 -6878.859,E2 -6878.859} C_VEL
LIN {X 0,Y 481.654,Z 290.486,A -85,B 0,C 180,E1 -6881.913,E2 -6881.913} C_VEL
LIN {X 0,Y 481.656,Z 290.484,A -85,B 0,C 180,E1 -6884.458,E2 -6884.458} C_VEL
LIN {X 0,Y 481.649,Z 290.488,A -85,B 0,C 180,E1 -6887.839,E2 -6887.839} C_VEL
LIN {X 0,Y 481.663,Z 290.483,A -85,B 0,C 180,E1 -6890.654,E2 -6890.654} C_VEL
LIN {X 0,Y 481.63,Z 290.494,A -85,B 0,C 180,E1 -6893.376,E2 -6893.376} C_VEL
LIN {X 0,Y 481.712,Z 290.483,A -85,B 0,C 180,E1 -6896.33,E2 -6896.33} C_VEL
LIN {X 0,Y 481.653,Z 290.49,A -85,B 0,C 180,E1 -6899.417,E2 -6899.417} C_VEL
LIN {X 0,Y 481.702,Z 290.486,A -85,B 0,C 180,E1 -6902.168,E2 -6902.168} C_VEL
LIN {X 0,Y 481.759,Z 290.606,A -85,B 0,C 180,E1 -6904.677,E2 -6904.677} C_VEL
LIN {X 0,Y 483.441,Z 299.973,A -85,B 0,C 180,E1 -6906.328,E2 -6906.328} C_VEL
LIN {X 0,Y 483.115,Z 313.724,A -85,B 0,C 180,E1 -6908.595,E2 -6908.595} C_VEL
LIN {X 0,Y 482.534,Z 334.398,A -85,B 0,C 180,E1 -6911.97,E2 -6911.97} C_VEL
LIN {X 0,Y 482.222,Z 343.66,A -85,B 0,C 180,E1 -6913.472,E2 -6913.472} C_VEL
LIN {X 0,Y 484.796,Z 361.613,A -85,B 0,C 180,E1 -6913.848,E2 -6913.848} C_VEL
LIN {X 0,Y 484.119,Z 452.252,A -85,B 0,C 180,E1 -6915.255,E2 -6915.255} C_VEL
LIN {X 0,Y 483.758,Z 465.495,A -85,B 0,C 180,E1 -6915.621,E2 -6915.621} C_VEL
LIN {X 0,Y 483.363,Z 478.813,A -85,B 0,C 180,E1 -6916.172,E2 -6916.172} C_VEL
LIN {X 0,Y 482.948,Z 491.29,A -85,B 0,C 180,E1 -6916.889,E2 -6916.889} C_VEL
LIN {X 0,Y 482.509,Z 502.324,A -85,B 0,C 180,E1 -6917.7,E2 -6917.7} C_VEL
LIN {X 0,Y 482.106,Z 512.714,A -85,B 0,C 180,E1 -6918.65,E2 -6918.65} C_VEL
LIN {X 0,Y 481.707,Z 522.04,A -85,B 0,C 180,E1 -6919.704,E2 -6919.704} C_VEL
LIN {X 0,Y 481.354,Z 531.105,A -85,B 0,C 180,E1 -6920.969,E2 -6920.969} C_VEL
LIN {X 0,Y 481.137,Z 538.411,A -85,B 0,C 180,E1 -6922.234,E2 -6922.234} C_VEL
LIN {X 0,Y 480.969,Z 544.374,A -85,B 0,C 180,E1 -6923.529,E2 -6923.529} C_VEL
LIN {X 0,Y 480.897,Z 549.471,A -85,B 0,C 180,E1 -6924.969,E2 -6924.969} C_VEL
LIN {X 0,Y 480.829,Z 551.8,A -85,B 0,C 180,E1 -6925.809,E2 -6925.809} C_VEL
LIN {X 0,Y 480.888,Z 553.697,A -85,B 0,C 180,E1 -6926.648,E2 -6926.648} C_VEL
LIN {X 0,Y 480.821,Z 556.132,A -85,B 0,C 180,E1 -6928.324,E2 -6928.324} C_VEL
LIN {X 0,Y 480.745,Z 556.979,A -85,B 0,C 180,E1 -6930,E2 -6930} C_VEL
LIN {X 0,Y 480.821,Z 556.161,A -85,B 0,C 180,E1 -6931.675,E2 -6931.675} C_VEL
LIN {X 0,Y 480.823,Z 555.161,A -85,B 0,C 180,E1 -6932.513,E2 -6932.513} C_VEL
LIN {X 0,Y 480.888,Z 553.755,A -85,B 0,C 180,E1 -6933.351,E2 -6933.351} C_VEL
LIN {X 0,Y 480.838,Z 550.792,A -85,B 0,C 180,E1 -6934.61,E2 -6934.61} C_VEL
LIN {X 0,Y 480.924,Z 546.781,A -85,B 0,C 180,E1 -6935.871,E2 -6935.871} C_VEL
LIN {X 0,Y 481.104,Z 540.6,A -85,B 0,C 180,E1 -6937.343,E2 -6937.343} C_VEL
LIN {X 0,Y 481.305,Z 533.851,A -85,B 0,C 180,E1 -6938.607,E2 -6938.607} C_VEL
LIN {X 0,Y 481.579,Z 525.473,A -85,B 0,C 180,E1 -6939.873,E2 -6939.873} C_VEL
LIN {X 0,Y 481.946,Z 516.852,A -85,B 0,C 180,E1 -6940.927,E2 -6940.927} C_VEL
LIN {X 0,Y 482.444,Z 506.233,A -85,B 0,C 180,E1 -6941.979,E2 -6941.979} C_VEL
LIN {X 0,Y 482.845,Z 494.89,A -85,B 0,C 180,E1 -6942.883,E2 -6942.883} C_VEL
LIN {X 0,Y 483.194,Z 484.035,A -85,B 0,C 180,E1 -6943.564,E2 -6943.564} C_VEL
LIN {X 0,Y 483.626,Z 471.956,A -85,B 0,C 180,E1 -6944.141,E2 -6944.141} C_VEL
LIN {X 0,Y 483.964,Z 458.876,A -85,B 0,C 180,E1 -6944.587,E2 -6944.587} C_VEL
LIN {X 0,Y 484.221,Z 446.477,A -85,B 0,C 180,E1 -6944.848,E2 -6944.848} C_VEL
LIN {X 0,Y 484.721,Z 360.253,A -85,B 0,C 180,E1 -6946.169,E2 -6946.169} C_VEL
LIN {X 0,Y 482.303,Z 344.334,A -85,B 0,C 180,E1 -6946.508,E2 -6946.508} C_VEL
LIN {X 0,Y 482.927,Z 326.131,A -85,B 0,C 180,E1 -6949.555,E2 -6949.555} C_VEL
LIN {X 0,Y 483.695,Z 307.927,A -85,B 0,C 180,E1 -6952.646,E2 -6952.646} C_VEL
LIN {X 0,Y 483.802,Z 301.434,A -85,B 0,C 180,E1 -6953.769,E2 -6953.769} C_VEL
LIN {X 0,Y 481.75,Z 290.479,A -85,B 0,C 180,E1 -6955.822,E2 -6955.822} C_VEL
LIN {X 0,Y 481.677,Z 290.481,A -85,B 0,C 180,E1 -6958.903,E2 -6958.903} C_VEL
LIN {X 0,Y 481.656,Z 290.492,A -85,B 0,C 180,E1 -6962.189,E2 -6962.189} C_VEL
LIN {X 0,Y 481.686,Z 290.481,A -85,B 0,C 180,E1 -6964.681,E2 -6964.681} C_VEL
LIN {X 0,Y 481.652,Z 290.487,A -85,B 0,C 180,E1 -6968.007,E2 -6968.007} C_VEL
LIN {X 0,Y 481.653,Z 290.484,A -85,B 0,C 180,E1 -6971.041,E2 -6971.041} C_VEL
LIN {X 0,Y 481.656,Z 290.491,A -85,B 0,C 180,E1 -6974.457,E2 -6974.457} C_VEL
LIN {X 0,Y 481.65,Z 290.484,A -85,B 0,C 180,E1 -6977.839,E2 -6977.839} C_VEL
LIN {X 0,Y 481.677,Z 290.489,A -85,B 0,C 180,E1 -6980.65,E2 -6980.65} C_VEL
LIN {X 0,Y 481.627,Z 290.487,A -85,B 0,C 180,E1 -6983.375,E2 -6983.375} C_VEL
LIN {X 0,Y 481.705,Z 290.479,A -85,B 0,C 180,E1 -6986.33,E2 -6986.33} C_VEL
LIN {X 0,Y 481.646,Z 290.486,A -85,B 0,C 180,E1 -6989.417,E2 -6989.417} C_VEL
LIN {X 0,Y 481.695,Z 290.478,A -85,B 0,C 180,E1 -6992.168,E2 -6992.168} C_VEL
LIN {X 0,Y 481.713,Z 290.483,A -85,B 0,C 180,E1 -6994.97,E2 -6994.97} C_VEL
LIN {X 0,Y 481.644,Z 290.485,A -85,B 0,C 180,E1 -6997.705,E2 -6997.705} C_VEL
LIN {X 0,Y 481.699,Z 290.477,A -85,B 0,C 180,E1 -7000.393,E2 -7000.393} C_VEL
LIN {X 0,Y 481.685,Z 290.484,A -85,B 0,C 180,E1 -7003.034,E2 -7003.034} C_VEL
LIN {X 0,Y 481.688,Z 290.483,A -85,B 0,C 180,E1 -7005.639,E2 -7005.639} C_VEL
LIN {X 0,Y 481.745,Z 290.471,A -85,B 0,C 180,E1 -7008.215,E2 -7008.215} C_VEL
LIN {X 0,Y 481.757,Z 290.477,A -85,B 0,C 180,E1 -7011.612,E2 -7011.612} C_VEL
LIN {X 0,Y 481.81,Z 290.465,A -85,B 0,C 180,E1 -7014.14,E2 -7014.14} C_VEL
LIN {X 0,Y 481.921,Z 290.456,A -85,B 0,C 180,E1 -7017.493,E2 -7017.493} C_VEL
LIN {X 0,Y 481.933,Z 290.453,A -85,B 0,C 180,E1 -7020,E2 -7020} C_VEL
LIN {X 0,Y 481.921,Z 290.45,A -85,B 0,C 180,E1 -7022.508,E2 -7022.508} C_VEL
LIN {X 0,Y 481.793,Z 290.474,A -85,B 0,C 180,E1 -7025.861,E2 -7025.861} C_VEL
LIN {X 0,Y 481.757,Z 290.473,A -85,B 0,C 180,E1 -7028.389,E2 -7028.389} C_VEL
LIN {X 0,Y 481.745,Z 290.476,A -85,B 0,C 180,E1 -7031.785,E2 -7031.785} C_VEL
LIN {X 0,Y 481.737,Z 290.472,A -85,B 0,C 180,E1 -7035.225,E2 -7035.225} C_VEL
LIN {X 0,Y 481.703,Z 290.479,A -85,B 0,C 180,E1 -7038.722,E2 -7038.722} C_VEL
LIN {X 0,Y 481.64,Z 290.484,A -85,B 0,C 180,E1 -7041.395,E2 -7041.395} C_VEL
LIN {X 0,Y 481.652,Z 290.488,A -85,B 0,C 180,E1 -7044.115,E2 -7044.115} C_VEL
LIN {X 0,Y 481.69,Z 290.479,A -85,B 0,C 180,E1 -7047.128,E2 -7047.128} C_VEL
LIN {X 0,Y 481.669,Z 290.481,A -85,B 0,C 180,E1 -7049.742,E2 -7049.742} C_VEL
LIN {X 0,Y 481.668,Z 290.489,A -85,B 0,C 180,E1 -7052.675,E2 -7052.675} C_VEL
LIN {X 0,Y 481.633,Z 290.485,A -85,B 0,C 180,E1 -7055.71,E2 -7055.71} C_VEL
LIN {X 0,Y 481.663,Z 290.489,A -85,B 0,C 180,E1 -7058.86,E2 -7058.86} C_VEL
LIN {X 0,Y 481.643,Z 290.484,A -85,B 0,C 180,E1 -7061.913,E2 -7061.913} C_VEL
LIN {X 0,Y 481.652,Z 290.485,A -85,B 0,C 180,E1 -7064.459,E2 -7064.459} C_VEL
LIN {X 0,Y 481.627,Z 290.486,A -85,B 0,C 180,E1 -7067.838,E2 -7067.838} C_VEL
LIN {X 0,Y 481.665,Z 290.49,A -85,B 0,C 180,E1 -7071.141,E2 -7071.141} C_VEL
LIN {X 0,Y 481.633,Z 290.485,A -85,B 0,C 180,E1 -7074.291,E2 -7074.291} C_VEL
LIN {X 0,Y 481.67,Z 290.489,A -85,B 0,C 180,E1 -7077.326,E2 -7077.326} C_VEL
LIN {X 0,Y 481.666,Z 290.481,A -85,B 0,C 180,E1 -7080.259,E2 -7080.259} C_VEL
LIN {X 0,Y 481.66,Z 290.486,A -85,B 0,C 180,E1 -7083.108,E2 -7083.108} C_VEL
LIN {X 0,Y 481.649,Z 290.487,A -85,B 0,C 180,E1 -7085.886,E2 -7085.886} C_VEL
LIN {X 0,Y 481.638,Z 290.488,A -85,B 0,C 180,E1 -7087.964,E2 -7087.964} C_VEL
LIN {X 0,Y 480.971,Z 290.569,A -85,B 0,C 180,E1 -7088.662,E2 -7088.662} C_VEL
LIN {X 0,Y 478.147,Z 290.926,A -85,B 0,C 180,E1 -7089.797,E2 -7089.797} C_VEL
LIN {X 0,Y 475.76,Z 291.222,A -85,B 0,C 180,E1 -7090.711,E2 -7090.711} C_VEL
LIN {X 0,Y 474.73,Z 291.35,A -85,B 0,C 180,E1 -7091.417,E2 -7091.417} C_VEL
LIN {X 0,Y 474.643,Z 291.361,A -85,B 0,C 180,E1 -7091.656,E2 -7091.656} C_VEL
LIN {X 0,Y 474.703,Z 291.349,A -85,B 0,C 180,E1 -7094.545,E2 -7094.545} C_VEL
LIN {X 0,Y 474.696,Z 291.355,A -85,B 0,C 180,E1 -7098.038,E2 -7098.038} C_VEL
LIN {X 0,Y 474.665,Z 291.356,A -85,B 0,C 180,E1 -7101.486,E2 -7101.486} C_VEL
LIN {X 0,Y 474.739,Z 291.353,A -85,B 0,C 180,E1 -7104.052,E2 -7104.052} C_VEL
LIN {X 0,Y 474.843,Z 291.332,A -85,B 0,C 180,E1 -7107.456,E2 -7107.456} C_VEL
LIN {X 0,Y 474.883,Z 291.332,A -85,B 0,C 180,E1 -7110,E2 -7110} C_VEL
LIN {X 0,Y 474.841,Z 291.336,A -85,B 0,C 180,E1 -7112.545,E2 -7112.545} C_VEL
LIN {X 0,Y 474.739,Z 291.348,A -85,B 0,C 180,E1 -7115.949,E2 -7115.949} C_VEL
LIN {X 0,Y 474.664,Z 291.361,A -85,B 0,C 180,E1 -7118.515,E2 -7118.515} C_VEL
LIN {X 0,Y 474.68,Z 291.353,A -85,B 0,C 180,E1 -7121.963,E2 -7121.963} C_VEL
LIN {X 0,Y 474.655,Z 291.355,A -85,B 0,C 180,E1 -7125.458,E2 -7125.458} C_VEL
LIN {X 0,Y 474.633,Z 291.366,A -85,B 0,C 180,E1 -7128.617,E2 -7128.617} C_VEL
LIN {X 0,Y 474.622,Z 291.365,A -85,B 0,C 180,E1 -7131.111,E2 -7131.111} C_VEL
LIN {X 0,Y 474.587,Z 291.37,A -85,B 0,C 180,E1 -7134.497,E2 -7134.497} C_VEL
LIN {X 0,Y 474.638,Z 291.511,A -85,B 0,C 180,E1 -7136.255,E2 -7136.255} C_VEL
LIN {X 0,Y 475.645,Z 297.458,A -85,B 0,C 180,E1 -7137.557,E2 -7137.557} C_VEL
LIN {X 0,Y 475.421,Z 308.816,A -85,B 0,C 180,E1 -7139.91,E2 -7139.91} C_VEL
LIN {X 0,Y 475.366,Z 310.872,A -85,B 0,C 180,E1 -7140.325,E2 -7140.325} C_VEL
LIN {X 0,Y 478.155,Z 325.609,A -85,B 0,C 180,E1 -7140.66,E2 -7140.66} C_VEL
LIN {X 0,Y 477.35,Z 418.059,A -85,B 0,C 180,E1 -7142.116,E2 -7142.116} C_VEL
LIN {X 0,Y 477.029,Z 431.434,A -85,B 0,C 180,E1 -7142.5,E2 -7142.5} C_VEL
LIN {X 0,Y 476.696,Z 444.468,A -85,B 0,C 180,E1 -7143.059,E2 -7143.059} C_VEL
LIN {X 0,Y 476.271,Z 455.904,A -85,B 0,C 180,E1 -7143.725,E2 -7143.725} C_VEL
LIN {X 0,Y 475.822,Z 466.884,A -85,B 0,C 180,E1 -7144.541,E2 -7144.541} C_VEL
LIN {X 0,Y 475.431,Z 477.497,A -85,B 0,C 180,E1 -7145.527,E2 -7145.527} C_VEL
LIN {X 0,Y 475.026,Z 486.244,A -85,B 0,C 180,E1 -7146.524,E2 -7146.524} C_VEL
LIN {X 0,Y 474.572,Z 495.46,A -85,B 0,C 180,E1 -7147.826,E2 -7147.826} C_VEL
LIN {X 0,Y 474.307,Z 502.328,A -85,B 0,C 180,E1 -7149.026,E2 -7149.026} C_VEL
LIN {X 0,Y 474.08,Z 508.783,A -85,B 0,C 180,E1 -7150.434,E2 -7150.434} C_VEL
LIN {X 0,Y 473.891,Z 513.779,A -85,B 0,C 180,E1 -7151.865,E2 -7151.865} C_VEL
LIN {X 0,Y 473.783,Z 517.615,A -85,B 0,C 180,E1 -7153.376,E2 -7153.376} C_VEL
LIN {X 0,Y 473.702,Z 519.708,A -85,B 0,C 180,E1 -7154.59,E2 -7154.59} C_VEL
LIN {X 0,Y 473.66,Z 520.963,A -85,B 0,C 180,E1 -7155.783,E2 -7155.783} C_VEL
LIN {X 0,Y 473.63,Z 521.418,A -85,B 0,C 180,E1 -7156.954,E2 -7156.954} C_VEL
LIN {X 0,Y 473.673,Z 521.104,A -85,B 0,C 180,E1 -7158.111,E2 -7158.111} C_VEL
LIN {X 0,Y 473.675,Z 520.11,A -85,B 0,C 180,E1 -7159.244,E2 -7159.244} C_VEL
LIN {X 0,Y 473.728,Z 518.194,A -85,B 0,C 180,E1 -7160.484,E2 -7160.484} C_VEL
LIN {X 0,Y 473.897,Z 515.113,A -85,B 0,C 180,E1 -7161.814,E2 -7161.814} C_VEL
LIN {X 0,Y 474.019,Z 510.727,A -85,B 0,C 180,E1 -7163.19,E2 -7163.19} C_VEL
LIN {X 0,Y 474.267,Z 504.39,A -85,B 0,C 180,E1 -7164.695,E2 -7164.695} C_VEL
LIN {X 0,Y 474.569,Z 497.207,A -85,B 0,C 180,E1 -7166.029,E2 -7166.029} C_VEL
LIN {X 0,Y 474.946,Z 489.457,A -85,B 0,C 180,E1 -7167.184,E2 -7167.184} C_VEL
LIN {X 0,Y 475.351,Z 479.936,A -85,B 0,C 180,E1 -7168.341,E2 -7168.341} C_VEL
LIN {X 0,Y 475.797,Z 469.538,A -85,B 0,C 180,E1 -7169.362,E2 -7169.362} C_VEL
LIN {X 0,Y 476.26,Z 458.406,A -85,B 0,C 180,E1 -7170.229,E2 -7170.229} C_VEL
LIN {X 0,Y 476.633,Z 446.748,A -85,B 0,C 180,E1 -7170.943,E2 -7170.943} C_VEL
LIN {X 0,Y 476.997,Z 434.489,A -85,B 0,C 180,E1 -7171.509,E2 -7171.509} C_VEL
LIN {X 0,Y 477.254,Z 422.178,A -85,B 0,C 180,E1 -7171.904,E2 -7171.904} C_VEL
LIN {X 0,Y 477.462,Z 405.392,A -85,B 0,C 180,E1 -7172.216,E2 -7172.216} C_VEL
LIN {X 0,Y 478.14,Z 324.728,A -85,B 0,C 180,E1 -7173.482,E2 -7173.482} C_VEL
LIN {X 0,Y 475.365,Z 310.142,A -85,B 0,C 180,E1 -7173.845,E2 -7173.845} C_VEL
LIN {X 0,Y 475.503,Z 296.037,A -85,B 0,C 180,E1 -7176.272,E2 -7176.272} C_VEL
LIN {X 0,Y 474.671,Z 291.362,A -85,B 0,C 180,E1 -7177.151,E2 -7177.151} C_VEL
LIN {X 0,Y 474.657,Z 291.359,A -85,B 0,C 180,E1 -7180.089,E2 -7180.089} C_VEL
LIN {X 0,Y 474.641,Z 291.363,A -85,B 0,C 180,E1 -7182.774,E2 -7182.774} C_VEL
LIN {X 0,Y 474.654,Z 291.365,A -85,B 0,C 180,E1 -7185.421,E2 -7185.421} C_VEL
LIN {X 0,Y 474.706,Z 291.352,A -85,B 0,C 180,E1 -7188.037,E2 -7188.037} C_VEL
LIN {X 0,Y 474.728,Z 291.353,A -85,B 0,C 180,E1 -7191.486,E2 -7191.486} C_VEL
LIN {X 0,Y 474.771,Z 291.347,A -85,B 0,C 180,E1 -7194.052,E2 -7194.052} C_VEL
LIN {X 0,Y 474.894,Z 291.33,A -85,B 0,C 180,E1 -7197.455,E2 -7197.455} C_VEL
LIN {X 0,Y 474.913,Z 291.329,A -85,B 0,C 180,E1 -7200,E2 -7200} C_VEL
LIN {X 0,Y 474.895,Z 291.327,A -85,B 0,C 180,E1 -7202.544,E2 -7202.544} C_VEL
LIN {X 0,Y 474.759,Z 291.349,A -85,B 0,C 180,E1 -7205.948,E2 -7205.948} C_VEL
LIN {X 0,Y 474.728,Z 291.35,A -85,B 0,C 180,E1 -7208.513,E2 -7208.513} C_VEL
LIN {X 0,Y 474.706,Z 291.353,A -85,B 0,C 180,E1 -7211.962,E2 -7211.962} C_VEL
LIN {X 0,Y 474.702,Z 291.35,A -85,B 0,C 180,E1 -7215.455,E2 -7215.455} C_VEL
LIN {X 0,Y 474.664,Z 291.357,A -85,B 0,C 180,E1 -7219.01,E2 -7219.01} C_VEL
LIN {X 0,Y 474.59,Z 291.362,A -85,B 0,C 180,E1 -7221.729,E2 -7221.729} C_VEL
LIN {X 0,Y 474.658,Z 291.358,A -85,B 0,C 180,E1 -7224.493,E2 -7224.493} C_VEL
LIN {X 0,Y 474.683,Z 291.35,A -85,B 0,C 180,E1 -7227.334,E2 -7227.334} C_VEL
LIN {X 0,Y 474.607,Z 291.362,A -85,B 0,C 180,E1 -7230.23,E2 -7230.23} C_VEL
LIN {X 0,Y 474.626,Z 291.364,A -85,B 0,C 180,E1 -7233.221,E2 -7233.221} C_VEL
LIN {X 0,Y 474.59,Z 291.364,A -85,B 0,C 180,E1 -7236.323,E2 -7236.323} C_VEL
LIN {X 0,Y 474.62,Z 291.363,A -85,B 0,C 180,E1 -7239.646,E2 -7239.646} C_VEL
LIN {X 0,Y 474.616,Z 291.365,A -85,B 0,C 180,E1 -7242.934,E2 -7242.934} C_VEL
LIN {X 0,Y 474.608,Z 291.364,A -85,B 0,C 180,E1 -7245.895,E2 -7245.895} C_VEL
LIN {X 0,Y 474.629,Z 291.361,A -85,B 0,C 180,E1 -7249.041,E2 -7249.041} C_VEL
LIN {X 0,Y 474.612,Z 291.368,A -85,B 0,C 180,E1 -7251.704,E2 -7251.704} C_VEL
LIN {X 0,Y 474.627,Z 291.363,A -85,B 0,C 180,E1 -7254.726,E2 -7254.726} C_VEL
LIN {X 0,Y 474.638,Z 291.368,A -85,B 0,C 180,E1 -7257.788,E2 -7257.788} C_VEL
LIN {X 0,Y 474.626,Z 291.362,A -85,B 0,C 180,E1 -7260.885,E2 -7260.885} C_VEL
LIN {X 0,Y 474.665,Z 291.364,A -85,B 0,C 180,E1 -7263.628,E2 -7263.628} C_VEL
LIN {X 0,Y 474.687,Z 291.425,A -85,B 0,C 180,E1 -7264.467,E2 -7264.467} C_VEL
LIN {X 0,Y 476.518,Z 301.55,A -85,B 0,C 180,E1 -7266.283,E2 -7266.283} C_VEL
LIN {X 0,Y 476.09,Z 316.761,A -85,B 0,C 180,E1 -7268.824,E2 -7268.824} C_VEL
LIN {X 0,Y 475.507,Z 335.428,A -85,B 0,C 180,E1 -7271.917,E2 -7271.917} C_VEL
LIN {X 0,Y 475.251,Z 343.437,A -85,B 0,C 180,E1 -7273.218,E2 -7273.218} C_VEL
LIN {X 0,Y 477.98,Z 362.652,A -85,B 0,C 180,E1 -7273.626,E2 -7273.626} C_VEL
LIN {X 0,Y 477.26,Z 451.955,A -85,B 0,C 180,E1 -7275.039,E2 -7275.039} C_VEL
LIN {X 0,Y 476.876,Z 465.176,A -85,B 0,C 180,E1 -7275.408,E2 -7275.408} C_VEL
LIN {X 0,Y 476.436,Z 478.482,A -85,B 0,C 180,E1 -7275.967,E2 -7275.967} C_VEL
LIN {X 0,Y 476.007,Z 490.957,A -85,B 0,C 180,E1 -7276.694,E2 -7276.694} C_VEL
LIN {X 0,Y 475.57,Z 501.907,A -85,B 0,C 180,E1 -7277.511,E2 -7277.511} C_VEL
LIN {X 0,Y 475.128,Z 512.397,A -85,B 0,C 180,E1 -7278.481,E2 -7278.481} C_VEL
LIN {X 0,Y 474.681,Z 521.734,A -85,B 0,C 180,E1 -7279.55,E2 -7279.55} C_VEL
LIN {X 0,Y 474.309,Z 530.81,A -85,B 0,C 180,E1 -7280.834,E2 -7280.834} C_VEL
LIN {X 0,Y 474.061,Z 538.124,A -85,B 0,C 180,E1 -7282.118,E2 -7282.118} C_VEL
LIN {X 0,Y 473.905,Z 543.06,A -85,B 0,C 180,E1 -7283.186,E2 -7283.186} C_VEL
LIN {X 0,Y 473.845,Z 547.862,A -85,B 0,C 180,E1 -7284.467,E2 -7284.467} C_VEL
LIN {X 0,Y 473.735,Z 551.53,A -85,B 0,C 180,E1 -7285.746,E2 -7285.746} C_VEL
LIN {X 0,Y 473.795,Z 553.429,A -85,B 0,C 180,E1 -7286.598,E2 -7286.598} C_VEL
LIN {X 0,Y 473.741,Z 554.85,A -85,B 0,C 180,E1 -7287.449,E2 -7287.449} C_VEL
LIN {X 0,Y 473.724,Z 555.866,A -85,B 0,C 180,E1 -7288.299,E2 -7288.299} C_VEL
LIN {X 0,Y 473.688,Z 556.49,A -85,B 0,C 180,E1 -7289.149,E2 -7289.149} C_VEL
LIN {X 0,Y 473.671,Z 556.715,A -85,B 0,C 180,E1 -7290,E2 -7290} C_VEL
LIN {X 0,Y 473.688,Z 556.502,A -85,B 0,C 180,E1 -7290.85,E2 -7290.85} C_VEL
LIN {X 0,Y 473.724,Z 555.895,A -85,B 0,C 180,E1 -7291.7,E2 -7291.7} C_VEL
LIN {X 0,Y 473.741,Z 554.894,A -85,B 0,C 180,E1 -7292.55,E2 -7292.55} C_VEL
LIN {X 0,Y 473.795,Z 553.483,A -85,B 0,C 180,E1 -7293.401,E2 -7293.401} C_VEL
LIN {X 0,Y 473.761,Z 550.516,A -85,B 0,C 180,E1 -7294.679,E2 -7294.679} C_VEL
LIN {X 0,Y 473.831,Z 546.497,A -85,B 0,C 180,E1 -7295.959,E2 -7295.959} C_VEL
LIN {X 0,Y 474.013,Z 540.306,A -85,B 0,C 180,E1 -7297.454,E2 -7297.454} C_VEL
LIN {X 0,Y 474.251,Z 533.547,A -85,B 0,C 180,E1 -7298.736,E2 -7298.736} C_VEL
LIN {X 0,Y 474.547,Z 525.155,A -85,B 0,C 180,E1 -7300.021,E2 -7300.021} C_VEL
LIN {X 0,Y 474.943,Z 516.515,A -85,B 0,C 180,E1 -7301.09,E2 -7301.09} C_VEL
LIN {X 0,Y 475.442,Z 506.131,A -85,B 0,C 180,E1 -7302.135,E2 -7302.135} C_VEL
LIN {X 0,Y 475.85,Z 495.591,A -85,B 0,C 180,E1 -7302.994,E2 -7302.994} C_VEL
LIN {X 0,Y 476.272,Z 483.61,A -85,B 0,C 180,E1 -7303.765,E2 -7303.765} C_VEL
LIN {X 0,Y 476.724,Z 471.482,A -85,B 0,C 180,E1 -7304.35,E2 -7304.35} C_VEL
LIN {X 0,Y 477.073,Z 458.322,A -85,B 0,C 180,E1 -7304.803,E2 -7304.803} C_VEL
LIN {X 0,Y 477.331,Z 445.656,A -85,B 0,C 180,E1 -7305.067,E2 -7305.067} C_VEL
LIN {X 0,Y 477.955,Z 361.515,A -85,B 0,C 180,E1 -7306.375,E2 -7306.375} C_VEL
LIN {X 0,Y 475.316,Z 344.051,A -85,B 0,C 180,E1 -7306.758,E2 -7306.758} C_VEL
LIN {X 0,Y 475.966,Z 325.871,A -85,B 0,C 180,E1 -7309.853,E2 -7309.853} C_VEL
LIN {X 0,Y 476.749,Z 308.967,A -85,B 0,C 180,E1 -7312.765,E2 -7312.765} C_VEL
LIN {X 0,Y 476.787,Z 302.241,A -85,B 0,C 180,E1 -7313.95,E2 -7313.95} C_VEL
LIN {X 0,Y 474.701,Z 291.357,A -85,B 0,C 180,E1 -7316.019,E2 -7316.019} C_VEL
LIN {X 0,Y 474.645,Z 291.363,A -85,B 0,C 180,E1 -7318.282,E2 -7318.282} C_VEL
LIN {X 0,Y 474.597,Z 291.362,A -85,B 0,C 180,E1 -7321.217,E2 -7321.217} C_VEL
LIN {X 0,Y 474.63,Z 291.366,A -85,B 0,C 180,E1 -7324.24,E2 -7324.24} C_VEL
LIN {X 0,Y 474.587,Z 291.363,A -85,B 0,C 180,E1 -7327.383,E2 -7327.383} C_VEL
LIN {X 0,Y 474.614,Z 291.364,A -85,B 0,C 180,E1 -7330.657,E2 -7330.657} C_VEL
LIN {X 0,Y 474.598,Z 291.361,A -85,B 0,C 180,E1 -7333.481,E2 -7333.481} C_VEL
LIN {X 0,Y 474.619,Z 291.368,A -85,B 0,C 180,E1 -7336.516,E2 -7336.516} C_VEL
LIN {X 0,Y 474.615,Z 291.36,A -85,B 0,C 180,E1 -7339.342,E2 -7339.342} C_VEL
LIN {X 0,Y 474.607,Z 291.36,A -85,B 0,C 180,E1 -7341.703,E2 -7341.703} C_VEL
LIN {X 0,Y 474.624,Z 291.367,A -85,B 0,C 180,E1 -7344.726,E2 -7344.726} C_VEL
LIN {X 0,Y 474.632,Z 291.357,A -85,B 0,C 180,E1 -7347.788,E2 -7347.788} C_VEL
LIN {X 0,Y 474.619,Z 291.367,A -85,B 0,C 180,E1 -7350.884,E2 -7350.884} C_VEL
LIN {X 0,Y 474.655,Z 291.356,A -85,B 0,C 180,E1 -7353.628,E2 -7353.628} C_VEL
LIN {X 0,Y 474.63,Z 291.36,A -85,B 0,C 180,E1 -7356.641,E2 -7356.641} C_VEL
LIN {X 0,Y 474.649,Z 291.355,A -85,B 0,C 180,E1 -7360.089,E2 -7360.089} C_VEL
LIN {X 0,Y 474.644,Z 291.358,A -85,B 0,C 180,E1 -7362.774,E2 -7362.774} C_VEL
LIN {X 0,Y 474.646,Z 291.363,A -85,B 0,C 180,E1 -7365.421,E2 -7365.421} C_VEL
LIN {X 0,Y 474.698,Z 291.35,A -85,B 0,C 180,E1 -7368.038,E2 -7368.038} C_VEL
LIN {X 0,Y 474.722,Z 291.355,A -85,B 0,C 180,E1 -7371.487,E2 -7371.487} C_VEL
LIN {X 0,Y 474.772,Z 291.342,A -85,B 0,C 180,E1 -7374.052,E2 -7374.052} C_VEL
